LIN {X -0.304,Y -476.004,Z 243.555,A 0.000,B 0.000,C 90.000,E1 135.972} C_DIS
LIN {X 0.127,Y -476.516,Z 243.548,A 0.000,B 0.000,C 90.000,E1 134.676} C_DIS
LIN {X -0.220,Y -476.712,Z 243.543,A 0.000,B 0.000,C 90.000,E1 133.785} C_DIS
LIN {X -0.220,Y -476.693,Z 243.538,A 0.000,B 0.000,C 90.000,E1 132.852} C_DIS
LIN {X -0.114,Y -476.300,Z 243.531,A 0.000,B 0.000,C 90.000,E1 131.595} C_DIS
LIN {X 0.027,Y -475.504,Z 243.524,A 0.000,B 0.000,C 90.000,E1 130.334} C_DIS
LIN {X 0.251,Y -474.323,Z 243.515,A 0.000,B 0.000,C 90.000,E1 128.749} C_DIS
LIN {X -0.093,Y -473.444,Z 243.510,A 0.000,B 0.000,C 90.000,E1 127.855} C_DIS
LIN {X 0.085,Y -471.985,Z 243.503,A 0.000,B 0.000,C 90.000,E1 126.583} C_DIS
LIN {X 0.086,Y -470.799,Z 243.498,A 0.000,B 0.000,C 90.000,E1 125.644} C_DIS
LIN {X -0.119,Y -467.941,Z 243.488,A 0.000,B 0.000,C 90.000,E1 123.785} C_DIS
LIN {X 0.106,Y -465.899,Z 243.481,A 0.000,B 0.000,C 90.000,E1 122.498} C_DIS
LIN {X -0.098,Y -463.753,Z 243.474,A 0.000,B 0.000,C 90.000,E1 121.258} C_DIS
LIN {X -0.050,Y -461.019,Z 243.465,A 0.000,B 0.000,C 90.000,E1 119.667} C_DIS
LIN {X -0.164,Y -457.610,Z 243.454,A 0.000,B 0.000,C 90.000,E1 117.769} C_DIS
LIN {X -0.057,Y -454.742,Z 243.445,A 0.000,B 0.000,C 90.000,E1 116.155} C_DIS
LIN {X -0.026,Y -450.753,Z 243.433,A 0.000,B 0.000,C 90.000,E1 113.898} C_DIS
LIN {X -0.037,Y -449.140,Z 243.428,A 0.000,B 0.000,C 90.000,E1 112.950} C_DIS
LIN {X -0.075,Y -449.131,Z 243.428,A 0.000,B 0.000,C 90.000,E1 112.950} C_DIS
LIN {X 0.220,Y -456.665,Z 243.411,A 0.000,B 0.000,C 90.000,E1 109.993} C_DIS
LIN {X -0.034,Y -457.470,Z 243.410,A 0.000,B 0.000,C 90.000,E1 109.704} C_DIS
LIN {X 0.067,Y -466.135,Z 243.386,A 0.000,B 0.000,C 90.000,E1 105.552} C_DIS
LIN {X -0.209,Y -467.704,Z 243.383,A 0.000,B 0.000,C 90.000,E1 104.954} C_DIS
LIN {X 0.216,Y -475.915,Z 243.357,A 0.000,B 0.000,C 90.000,E1 100.197} C_DIS
LIN {X 0.055,Y -476.355,Z 243.355,A 0.000,B 0.000,C 90.000,E1 99.905} C_DIS
LIN {X 0.012,Y -481.875,Z 243.331,A 0.000,B 0.000,C 90.000,E1 95.568} C_DIS
LIN {X -0.141,Y -482.193,Z 243.329,A 0.000,B 0.000,C 90.000,E1 95.277} C_DIS
LIN {X -0.207,Y -485.365,Z 243.305,A 0.000,B 0.000,C 90.000,E1 90.974} C_DIS
LIN {X 0.102,Y -485.531,Z 243.304,A 0.000,B 0.000,C 90.000,E1 90.630} C_DIS
LIN {X -0.175,Y -486.345,Z 243.281,A 0.000,B 0.000,C 90.000,E1 86.674} C_DIS
LIN {X -0.041,Y -486.268,Z 243.278,A 0.000,B 0.000,C 90.000,E1 86.045} C_DIS
LIN {X 0.158,Y -484.694,Z 243.254,A 0.000,B 0.000,C 90.000,E1 81.724} C_DIS
LIN {X 0.026,Y -484.535,Z 243.252,A 0.000,B 0.000,C 90.000,E1 81.432} C_DIS
LIN {X -0.104,Y -480.473,Z 243.227,A 0.000,B 0.000,C 90.000,E1 76.825} C_DIS
LIN {X -0.207,Y -474.232,Z 243.201,A 0.000,B 0.000,C 90.000,E1 72.181} C_DIS
LIN {X 0.212,Y -473.736,Z 243.199,A 0.000,B 0.000,C 90.000,E1 71.819} C_DIS
LIN {X -0.275,Y -466.180,Z 243.175,A 0.000,B 0.000,C 90.000,E1 67.486} C_DIS
LIN {X 0.276,Y -465.753,Z 243.173,A 0.000,B 0.000,C 90.000,E1 67.102} C_DIS
LIN {X 0.046,Y -464.164,Z 243.169,A 0.000,B 0.000,C 90.000,E1 66.410} C_DIS
LIN {X 0.006,Y -464.156,Z 243.169,A 0.000,B 0.000,C 90.000,E1 66.410} C_DIS
LIN {X 0.084,Y -467.157,Z 243.162,A 0.000,B 0.000,C 90.000,E1 65.229} C_DIS
LIN {X 0.048,Y -470.372,Z 243.155,A 0.000,B 0.000,C 90.000,E1 63.973} C_DIS
LIN {X -0.028,Y -475.351,Z 243.145,A 0.000,B 0.000,C 90.000,E1 62.103} C_DIS
LIN {X 0.024,Y -481.156,Z 243.133,A 0.000,B 0.000,C 90.000,E1 59.921} C_DIS
LIN {X 0.004,Y -486.185,Z 243.123,A 0.000,B 0.000,C 90.000,E1 58.074} C_DIS
LIN {X -0.048,Y -490.388,Z 243.114,A 0.000,B 0.000,C 90.000,E1 56.548} C_DIS
LIN {X -0.011,Y -494.338,Z 243.106,A 0.000,B 0.000,C 90.000,E1 55.022} C_DIS
LIN {X -0.174,Y -497.233,Z 243.099,A 0.000,B 0.000,C 90.000,E1 53.829} C_DIS
LIN {X -0.174,Y -499.342,Z 243.094,A 0.000,B 0.000,C 90.000,E1 52.924} C_DIS
LIN {X 0.026,Y -501.806,Z 243.087,A 0.000,B 0.000,C 90.000,E1 51.698} C_DIS
LIN {X -0.131,Y -504.092,Z 243.081,A 0.000,B 0.000,C 90.000,E1 50.517} C_DIS
LIN {X -0.039,Y -506.583,Z 243.072,A 0.000,B 0.000,C 90.000,E1 49.013} C_DIS
LIN {X -0.178,Y -508.187,Z 243.066,A 0.000,B 0.000,C 90.000,E1 47.838} C_DIS
LIN {X -0.048,Y -508.957,Z 243.062,A 0.000,B 0.000,C 90.000,E1 47.229} C_DIS
LIN {X -0.149,Y -510.048,Z 243.056,A 0.000,B 0.000,C 90.000,E1 46.053} C_DIS
LIN {X 0.120,Y -510.862,Z 243.049,A 0.000,B 0.000,C 90.000,E1 44.838} C_DIS
LIN {X 0.048,Y -511.450,Z 243.043,A 0.000,B 0.000,C 90.000,E1 43.662} C_DIS
LIN {X 0.083,Y -511.654,Z 243.038,A 0.000,B 0.000,C 90.000,E1 42.771} C_DIS
LIN {X 0.018,Y -511.694,Z 243.031,A 0.000,B 0.000,C 90.000,E1 41.595} C_DIS
LIN {X -0.001,Y -511.374,Z 243.025,A 0.000,B 0.000,C 90.000,E1 40.415} C_DIS
LIN {X 0.309,Y -510.843,Z 243.018,A 0.000,B 0.000,C 90.000,E1 39.197} C_DIS
LIN {X 0.279,Y -509.901,Z 243.011,A 0.000,B 0.000,C 90.000,E1 38.016} C_DIS
LIN {X -0.079,Y -508.670,Z 243.005,A 0.000,B 0.000,C 90.000,E1 36.870} C_DIS
LIN {X -0.138,Y -506.605,Z 242.997,A 0.000,B 0.000,C 90.000,E1 35.391} C_DIS
LIN {X 0.072,Y -503.848,Z 242.987,A 0.000,B 0.000,C 90.000,E1 33.579} C_DIS
LIN {X 0.231,Y -500.339,Z 242.975,A 0.000,B 0.000,C 90.000,E1 31.465} C_DIS
LIN {X 0.059,Y -496.727,Z 242.962,A 0.000,B 0.000,C 90.000,E1 29.077} C_DIS
LIN {X -0.146,Y -492.657,Z 242.943,A 0.000,B 0.000,C 90.000,E1 25.771} C_DIS
LIN {X -0.140,Y -490.689,Z 242.931,A 0.000,B 0.000,C 90.000,E1 23.643} C_DIS
LIN {X 0.113,Y -488.478,Z 242.918,A 0.000,B 0.000,C 90.000,E1 21.173} C_DIS
LIN {X 0.135,Y -486.122,Z 242.902,A 0.000,B 0.000,C 90.000,E1 18.417} C_DIS
LIN {X 0.208,Y -484.424,Z 242.891,A 0.000,B 0.000,C 90.000,E1 16.260} C_DIS
LIN {X 0.101,Y -482.861,Z 242.879,A 0.000,B 0.000,C 90.000,E1 14.120} C_DIS
LIN {X -0.140,Y -481.824,Z 242.868,A 0.000,B 0.000,C 90.000,E1 12.299} C_DIS
LIN {X -0.164,Y -480.841,Z 242.856,A 0.000,B 0.000,C 90.000,E1 10.141} C_DIS
LIN {X 0.184,Y -480.149,Z 242.844,A 0.000,B 0.000,C 90.000,E1 7.936} C_DIS
LIN {X -0.241,Y -479.561,Z 242.831,A 0.000,B 0.000,C 90.000,E1 5.511} C_DIS
LIN {X 0.214,Y -479.518,Z 242.817,A 0.000,B 0.000,C 90.000,E1 2.980} C_DIS
LIN {X 0.105,Y -479.572,Z 242.812,A 0.000,B 0.000,C 90.000,E1 2.064} C_DIS
LIN {X 0.182,Y -480.137,Z 242.799,A 0.000,B 0.000,C 90.000,E1 359.771} C_DIS
LIN {X -0.082,Y -481.724,Z 242.783,A 0.000,B 0.000,C 90.000,E1 357.020} C_DIS
LIN {X 0.127,Y -483.318,Z 242.771,A 0.000,B 0.000,C 90.000,E1 354.837} C_DIS
LIN {X -0.041,Y -488.218,Z 242.748,A 0.000,B 0.000,C 90.000,E1 350.557} C_DIS
LIN {X 0.050,Y -492.322,Z 242.736,A 0.000,B 0.000,C 90.000,E1 348.409} C_DIS
LIN {X -0.131,Y -501.097,Z 242.717,A 0.000,B 0.000,C 90.000,E1 345.102} C_DIS
LIN {X 0.190,Y -506.043,Z 242.707,A 0.000,B 0.000,C 90.000,E1 343.268} C_DIS
LIN {X -0.058,Y -511.034,Z 242.697,A 0.000,B 0.000,C 90.000,E1 341.511} C_DIS
LIN {X -0.173,Y -521.016,Z 242.679,A 0.000,B 0.000,C 90.000,E1 338.284} C_DIS
LIN {X -0.192,Y -527.006,Z 242.670,A 0.000,B 0.000,C 90.000,E1 336.538} C_DIS
LIN {X -0.083,Y -533.082,Z 242.660,A 0.000,B 0.000,C 90.000,E1 334.793} C_DIS
LIN {X -0.107,Y -539.365,Z 242.650,A 0.000,B 0.000,C 90.000,E1 333.076} C_DIS
LIN {X -0.230,Y -545.756,Z 242.641,A 0.000,B 0.000,C 90.000,E1 331.385} C_DIS
LIN {X -0.216,Y -550.002,Z 242.635,A 0.000,B 0.000,C 90.000,E1 330.255} C_DIS
LIN {X 0.110,Y -555.145,Z 242.627,A 0.000,B 0.000,C 90.000,E1 328.820} C_DIS
LIN {X -0.088,Y -564.318,Z 242.613,A 0.000,B 0.000,C 90.000,E1 326.342} C_DIS
LIN {X 0.078,Y -571.677,Z 242.602,A 0.000,B 0.000,C 90.000,E1 324.402} C_DIS
LIN {X -0.167,Y -575.756,Z 242.596,A 0.000,B 0.000,C 90.000,E1 323.336} C_DIS
LIN {X -0.200,Y -580.262,Z 242.589,A 0.000,B 0.000,C 90.000,E1 321.984} C_DIS
LIN {X -0.276,Y -591.820,Z 242.571,A 0.000,B 0.000,C 90.000,E1 318.771} C_DIS
LIN {X 0.056,Y -596.053,Z 242.565,A 0.000,B 0.000,C 90.000,E1 317.676} C_DIS
LIN {X 0.042,Y -600.105,Z 242.559,A 0.000,B 0.000,C 90.000,E1 316.620} C_DIS
LIN {X 0.055,Y -603.953,Z 242.553,A 0.000,B 0.000,C 90.000,E1 315.567} C_DIS
LIN {X -0.066,Y -608.129,Z 242.546,A 0.000,B 0.000,C 90.000,E1 314.271} C_DIS
LIN {X 0.237,Y -610.253,Z 242.542,A 0.000,B 0.000,C 90.000,E1 313.461} C_DIS
LIN {X -0.035,Y -612.686,Z 242.536,A 0.000,B 0.000,C 90.000,E1 312.447} C_DIS
LIN {X 0.182,Y -614.592,Z 242.530,A 0.000,B 0.000,C 90.000,E1 311.391} C_DIS
LIN {X -0.036,Y -616.293,Z 242.524,A 0.000,B 0.000,C 90.000,E1 310.378} C_DIS
LIN {X 0.398,Y -617.459,Z 242.520,A 0.000,B 0.000,C 90.000,E1 309.564} C_DIS
LIN {X 0.291,Y -618.870,Z 242.514,A 0.000,B 0.000,C 90.000,E1 308.543} C_DIS
LIN {X 0.205,Y -620.140,Z 242.509,A 0.000,B 0.000,C 90.000,E1 307.523} C_DIS
LIN {X -0.193,Y -620.790,Z 242.504,A 0.000,B 0.000,C 90.000,E1 306.790} C_DIS
LIN {X -0.305,Y -621.404,Z 242.497,A 0.000,B 0.000,C 90.000,E1 305.518} C_DIS
LIN {X -0.197,Y -621.670,Z 242.493,A 0.000,B 0.000,C 90.000,E1 304.739} C_DIS
LIN {X 0.426,Y -621.842,Z 242.489,A 0.000,B 0.000,C 90.000,E1 303.913} C_DIS
LIN {X -0.348,Y -621.735,Z 242.483,A 0.000,B 0.000,C 90.000,E1 302.959} C_DIS
LIN {X 0.275,Y -621.168,Z 242.479,A 0.000,B 0.000,C 90.000,E1 302.133} C_DIS
LIN {X 0.018,Y -620.148,Z 242.473,A 0.000,B 0.000,C 90.000,E1 301.131} C_DIS
LIN {X 0.297,Y -619.048,Z 242.469,A 0.000,B 0.000,C 90.000,E1 300.335} C_DIS
LIN {X 0.010,Y -617.161,Z 242.463,A 0.000,B 0.000,C 90.000,E1 299.333} C_DIS
LIN {X -0.043,Y -615.539,Z 242.459,A 0.000,B 0.000,C 90.000,E1 298.565} C_DIS
LIN {X 0.129,Y -612.600,Z 242.452,A 0.000,B 0.000,C 90.000,E1 297.257} C_DIS
LIN {X 0.002,Y -609.954,Z 242.446,A 0.000,B 0.000,C 90.000,E1 296.232} C_DIS
LIN {X -0.210,Y -606.449,Z 242.439,A 0.000,B 0.000,C 90.000,E1 294.951} C_DIS
LIN {X -0.249,Y -602.264,Z 242.430,A 0.000,B 0.000,C 90.000,E1 293.387} C_DIS
LIN {X -0.218,Y -597.176,Z 242.418,A 0.000,B 0.000,C 90.000,E1 291.280} C_DIS
LIN {X 0.127,Y -592.982,Z 242.408,A 0.000,B 0.000,C 90.000,E1 289.396} C_DIS
LIN {X 0.188,Y -588.928,Z 242.398,A 0.000,B 0.000,C 90.000,E1 287.528} C_DIS
LIN {X 0.059,Y -584.239,Z 242.384,A 0.000,B 0.000,C 90.000,E1 285.134} C_DIS
LIN {X -0.183,Y -580.544,Z 242.372,A 0.000,B 0.000,C 90.000,E1 283.008} C_DIS
LIN {X -0.011,Y -576.449,Z 242.356,A 0.000,B 0.000,C 90.000,E1 280.018} C_DIS
LIN {X 0.186,Y -573.364,Z 242.339,A 0.000,B 0.000,C 90.000,E1 277.011} C_DIS
LIN {X 0.173,Y -571.959,Z 242.329,A 0.000,B 0.000,C 90.000,E1 275.106} C_DIS
LIN {X 0.208,Y -570.930,Z 242.297,A 0.000,B 0.000,C 90.000,E1 269.370} C_DIS
LIN {X -0.192,Y -574.912,Z 242.265,A 0.000,B 0.000,C 90.000,E1 263.685} C_DIS
LIN {X 0.272,Y -577.835,Z 242.251,A 0.000,B 0.000,C 90.000,E1 261.197} C_DIS
LIN {X 0.008,Y -581.772,Z 242.236,A 0.000,B 0.000,C 90.000,E1 258.522} C_DIS
LIN {X -0.055,Y -584.686,Z 242.226,A 0.000,B 0.000,C 90.000,E1 256.645} C_DIS
LIN {X 0.098,Y -585.933,Z 242.221,A 0.000,B 0.000,C 90.000,E1 255.825} C_DIS
LIN {X -0.236,Y -587.935,Z 242.214,A 0.000,B 0.000,C 90.000,E1 254.519} C_DIS
LIN {X -0.053,Y -589.315,Z 242.208,A 0.000,B 0.000,C 90.000,E1 253.433} C_DIS
LIN {X -0.121,Y -589.865,Z 242.205,A 0.000,B 0.000,C 90.000,E1 252.906} C_DIS
LIN {X -0.332,Y -590.543,Z 242.201,A 0.000,B 0.000,C 90.000,E1 252.127} C_DIS
LIN {X -0.109,Y -590.938,Z 242.195,A 0.000,B 0.000,C 90.000,E1 251.040} C_DIS
LIN {X 0.319,Y -591.095,Z 242.189,A 0.000,B 0.000,C 90.000,E1 249.934} C_DIS
LIN {X -0.007,Y -591.001,Z 242.183,A 0.000,B 0.000,C 90.000,E1 248.901} C_DIS
LIN {X -0.012,Y -590.558,Z 242.178,A 0.000,B 0.000,C 90.000,E1 248.103} C_DIS
LIN {X -0.026,Y -589.930,Z 242.174,A 0.000,B 0.000,C 90.000,E1 247.305} C_DIS
LIN {X 0.072,Y -588.643,Z 242.168,A 0.000,B 0.000,C 90.000,E1 246.230} C_DIS
LIN {X 0.273,Y -587.450,Z 242.164,A 0.000,B 0.000,C 90.000,E1 245.409} C_DIS
LIN {X 0.092,Y -585.402,Z 242.158,A 0.000,B 0.000,C 90.000,E1 244.357} C_DIS
LIN {X 0.257,Y -582.356,Z 242.150,A 0.000,B 0.000,C 90.000,E1 242.999} C_DIS
LIN {X -0.135,Y -578.999,Z 242.143,A 0.000,B 0.000,C 90.000,E1 241.691} C_DIS
LIN {X 0.076,Y -576.071,Z 242.137,A 0.000,B 0.000,C 90.000,E1 240.589} C_DIS
LIN {X -0.101,Y -573.711,Z 242.132,A 0.000,B 0.000,C 90.000,E1 239.793} C_DIS
LIN {X 0.255,Y -568.612,Z 242.123,A 0.000,B 0.000,C 90.000,E1 238.122} C_DIS
LIN {X -0.094,Y -564.190,Z 242.115,A 0.000,B 0.000,C 90.000,E1 236.786} C_DIS
LIN {X 0.047,Y -557.249,Z 242.103,A 0.000,B 0.000,C 90.000,E1 234.562} C_DIS
LIN {X -0.003,Y -552.836,Z 242.095,A 0.000,B 0.000,C 90.000,E1 233.176} C_DIS
LIN {X 0.027,Y -547.568,Z 242.086,A 0.000,B 0.000,C 90.000,E1 231.492} C_DIS
LIN {X -0.235,Y -542.222,Z 242.077,A 0.000,B 0.000,C 90.000,E1 229.828} C_DIS
LIN {X 0.163,Y -536.815,Z 242.067,A 0.000,B 0.000,C 90.000,E1 228.081} C_DIS
LIN {X 0.036,Y -531.322,Z 242.058,A 0.000,B 0.000,C 90.000,E1 226.377} C_DIS
LIN {X 0.198,Y -526.688,Z 242.050,A 0.000,B 0.000,C 90.000,E1 224.919} C_DIS
LIN {X -0.164,Y -521.139,Z 242.040,A 0.000,B 0.000,C 90.000,E1 223.218} C_DIS
LIN {X 0.033,Y -514.869,Z 242.029,A 0.000,B 0.000,C 90.000,E1 221.148} C_DIS
LIN {X 0.129,Y -508.712,Z 242.017,A 0.000,B 0.000,C 90.000,E1 219.072} C_DIS
LIN {X 0.060,Y -502.784,Z 242.006,A 0.000,B 0.000,C 90.000,E1 216.996} C_DIS
LIN {X 0.160,Y -497.674,Z 241.996,A 0.000,B 0.000,C 90.000,E1 215.185} C_DIS
LIN {X -0.109,Y -493.403,Z 241.987,A 0.000,B 0.000,C 90.000,E1 213.706} C_DIS
LIN {X -0.072,Y -488.405,Z 241.977,A 0.000,B 0.000,C 90.000,E1 211.878} C_DIS
LIN {X -0.168,Y -482.790,Z 241.965,A 0.000,B 0.000,C 90.000,E1 209.745} C_DIS
LIN {X -0.152,Y -474.126,Z 241.945,A 0.000,B 0.000,C 90.000,E1 206.027} C_DIS
LIN {X -0.023,Y -469.618,Z 241.932,A 0.000,B 0.000,C 90.000,E1 203.823} C_DIS
LIN {X -0.251,Y -462.865,Z 241.911,A 0.000,B 0.000,C 90.000,E1 200.066} C_DIS
LIN {X -0.040,Y -458.061,Z 241.894,A 0.000,B 0.000,C 90.000,E1 196.858} C_DIS
LIN {X 0.143,Y -454.256,Z 241.878,A 0.000,B 0.000,C 90.000,E1 193.953} C_DIS
LIN {X 0.059,Y -452.251,Z 241.869,A 0.000,B 0.000,C 90.000,E1 192.355} C_DIS
LIN {X -0.106,Y -449.238,Z 241.854,A 0.000,B 0.000,C 90.000,E1 189.792} C_DIS
LIN {X 0.010,Y -446.505,Z 241.840,A 0.000,B 0.000,C 90.000,E1 187.182} C_DIS
LIN {X 0.200,Y -444.448,Z 241.827,A 0.000,B 0.000,C 90.000,E1 184.878} C_DIS
LIN {X -0.109,Y -443.337,Z 241.820,A 0.000,B 0.000,C 90.000,E1 183.612} C_DIS
LIN {X -0.022,Y -442.321,Z 241.813,A 0.000,B 0.000,C 90.000,E1 182.293} C_DIS
LIN {X 0.169,Y -441.174,Z 241.804,A 0.000,B 0.000,C 90.000,E1 180.630} C_DIS
LIN {X -0.190,Y -439.660,Z 241.789,A 0.000,B 0.000,C 90.000,E1 178.051} C_DIS
LIN {X 0.101,Y -438.687,Z 241.771,A 0.000,B 0.000,C 90.000,E1 174.723} C_DIS
LIN {X -0.213,Y -438.624,Z 241.751,A 0.000,B 0.000,C 90.000,E1 171.141} C_DIS
LIN {X 0.102,Y -439.157,Z 241.736,A 0.000,B 0.000,C 90.000,E1 168.465} C_DIS
LIN {X -0.031,Y -440.655,Z 241.716,A 0.000,B 0.000,C 90.000,E1 164.866} C_DIS
LIN {X 0.008,Y -441.997,Z 241.701,A 0.000,B 0.000,C 90.000,E1 162.236} C_DIS
LIN {X 0.086,Y -443.455,Z 241.689,A 0.000,B 0.000,C 90.000,E1 159.934} C_DIS
LIN {X 0.076,Y -446.041,Z 241.672,A 0.000,B 0.000,C 90.000,E1 156.997} C_DIS
LIN {X 0.106,Y -448.492,Z 241.660,A 0.000,B 0.000,C 90.000,E1 154.717} C_DIS
LIN {X -0.112,Y -451.766,Z 241.645,A 0.000,B 0.000,C 90.000,E1 152.153} C_DIS
LIN {X 0.095,Y -455.084,Z 241.633,A 0.000,B 0.000,C 90.000,E1 149.871} C_DIS
LIN {X -0.173,Y -458.625,Z 241.620,A 0.000,B 0.000,C 90.000,E1 147.661} C_DIS
LIN {X 0.151,Y -462.336,Z 241.608,A 0.000,B 0.000,C 90.000,E1 145.388} C_DIS
LIN {X -0.075,Y -464.957,Z 241.599,A 0.000,B 0.000,C 90.000,E1 143.829} C_DIS
LIN {X -0.255,Y -467.359,Z 241.590,A 0.000,B 0.000,C 90.000,E1 142.271} C_DIS
LIN {X -0.048,Y -470.004,Z 241.580,A 0.000,B 0.000,C 90.000,E1 140.356} C_DIS
LIN {X 0.082,Y -471.957,Z 241.571,A 0.000,B 0.000,C 90.000,E1 138.771} C_DIS
LIN {X -0.199,Y -473.178,Z 241.564,A 0.000,B 0.000,C 90.000,E1 137.553} C_DIS
LIN {X -0.144,Y -474.125,Z 241.557,A 0.000,B 0.000,C 90.000,E1 136.296} C_DIS
LIN {X 0.054,Y -474.411,Z 241.554,A 0.000,B 0.000,C 90.000,E1 135.648} C_DIS
LIN {X 0.256,Y -474.787,Z 241.550,A 0.000,B 0.000,C 90.000,E1 135.000} C_DIS
LIN {X -0.007,Y -475.074,Z 241.543,A 0.000,B 0.000,C 90.000,E1 133.785} C_DIS
LIN {X -0.026,Y -475.093,Z 241.538,A 0.000,B 0.000,C 90.000,E1 132.852} C_DIS
LIN {X 0.055,Y -474.641,Z 241.531,A 0.000,B 0.000,C 90.000,E1 131.595} C_DIS
LIN {X 0.260,Y -473.640,Z 241.523,A 0.000,B 0.000,C 90.000,E1 130.011} C_DIS
LIN {X -0.304,Y -472.672,Z 241.516,A 0.000,B 0.000,C 90.000,E1 128.830} C_DIS
LIN {X 0.000,Y -471.795,Z 241.510,A 0.000,B 0.000,C 90.000,E1 127.855} C_DIS
LIN {X 0.152,Y -470.389,Z 241.503,A 0.000,B 0.000,C 90.000,E1 126.583} C_DIS
LIN {X -0.095,Y -468.779,Z 241.496,A 0.000,B 0.000,C 90.000,E1 125.358} C_DIS
LIN {X 0.043,Y -465.891,Z 241.486,A 0.000,B 0.000,C 90.000,E1 123.452} C_DIS
LIN {X -0.154,Y -463.815,Z 241.479,A 0.000,B 0.000,C 90.000,E1 122.212} C_DIS
LIN {X 0.002,Y -461.640,Z 241.472,A 0.000,B 0.000,C 90.000,E1 120.924} C_DIS
LIN {X 0.008,Y -458.916,Z 241.463,A 0.000,B 0.000,C 90.000,E1 119.333} C_DIS
LIN {X 0.140,Y -456.050,Z 241.454,A 0.000,B 0.000,C 90.000,E1 117.719} C_DIS
LIN {X 0.110,Y -452.565,Z 241.443,A 0.000,B 0.000,C 90.000,E1 115.796} C_DIS
LIN {X -0.137,Y -448.627,Z 241.431,A 0.000,B 0.000,C 90.000,E1 113.567} C_DIS
LIN {X -0.056,Y -448.249,Z 241.430,A 0.000,B 0.000,C 90.000,E1 113.334} C_DIS
LIN {X -0.096,Y -448.253,Z 241.430,A 0.000,B 0.000,C 90.000,E1 113.334} C_DIS
LIN {X 0.025,Y -456.735,Z 241.411,A 0.000,B 0.000,C 90.000,E1 109.993} C_DIS
LIN {X -0.074,Y -457.513,Z 241.409,A 0.000,B 0.000,C 90.000,E1 109.685} C_DIS
LIN {X -0.129,Y -466.192,Z 241.386,A 0.000,B 0.000,C 90.000,E1 105.552} C_DIS
LIN {X 0.048,Y -467.758,Z 241.383,A 0.000,B 0.000,C 90.000,E1 104.898} C_DIS
LIN {X 0.020,Y -475.965,Z 241.357,A 0.000,B 0.000,C 90.000,E1 100.197} C_DIS
LIN {X 0.169,Y -476.677,Z 241.353,A 0.000,B 0.000,C 90.000,E1 99.557} C_DIS
LIN {X -0.186,Y -481.913,Z 241.331,A 0.000,B 0.000,C 90.000,E1 95.568} C_DIS
LIN {X 0.142,Y -482.202,Z 241.329,A 0.000,B 0.000,C 90.000,E1 95.220} C_DIS
LIN {X 0.080,Y -485.389,Z 241.305,A 0.000,B 0.000,C 90.000,E1 90.917} C_DIS
LIN {X -0.096,Y -485.529,Z 241.303,A 0.000,B 0.000,C 90.000,E1 90.630} C_DIS
LIN {X 0.113,Y -486.357,Z 241.281,A 0.000,B 0.000,C 90.000,E1 86.617} C_DIS
LIN {X -0.063,Y -486.368,Z 241.280,A 0.000,B 0.000,C 90.000,E1 86.331} C_DIS
LIN {X -0.074,Y -485.858,Z 241.275,A 0.000,B 0.000,C 90.000,E1 85.412} C_DIS
LIN {X -0.039,Y -484.692,Z 241.254,A 0.000,B 0.000,C 90.000,E1 81.724} C_DIS
LIN {X -0.171,Y -484.506,Z 241.252,A 0.000,B 0.000,C 90.000,E1 81.432} C_DIS
LIN {X 0.167,Y -480.439,Z 241.227,A 0.000,B 0.000,C 90.000,E1 76.769} C_DIS
LIN {X 0.049,Y -474.209,Z 241.201,A 0.000,B 0.000,C 90.000,E1 72.127} C_DIS
LIN {X -0.017,Y -473.050,Z 241.197,A 0.000,B 0.000,C 90.000,E1 71.511} C_DIS
LIN {X 0.081,Y -465.722,Z 241.173,A 0.000,B 0.000,C 90.000,E1 67.102} C_DIS
LIN {X -0.052,Y -463.440,Z 241.167,A 0.000,B 0.000,C 90.000,E1 66.102} C_DIS
LIN {X -0.092,Y -463.437,Z 241.167,A 0.000,B 0.000,C 90.000,E1 66.102} C_DIS
LIN {X -0.056,Y -467.282,Z 241.159,A 0.000,B 0.000,C 90.000,E1 64.588} C_DIS
LIN {X 0.174,Y -473.040,Z 241.147,A 0.000,B 0.000,C 90.000,E1 62.359} C_DIS
LIN {X -0.025,Y -477.955,Z 241.136,A 0.000,B 0.000,C 90.000,E1 60.511} C_DIS
LIN {X -0.120,Y -481.302,Z 241.129,A 0.000,B 0.000,C 90.000,E1 59.282} C_DIS
LIN {X 0.105,Y -486.372,Z 241.119,A 0.000,B 0.000,C 90.000,E1 57.406} C_DIS
LIN {X -0.187,Y -489.686,Z 241.112,A 0.000,B 0.000,C 90.000,E1 56.215} C_DIS
LIN {X -0.016,Y -492.807,Z 241.105,A 0.000,B 0.000,C 90.000,E1 54.975} C_DIS
LIN {X -0.055,Y -496.411,Z 241.097,A 0.000,B 0.000,C 90.000,E1 53.463} C_DIS
LIN {X -0.063,Y -498.422,Z 241.092,A 0.000,B 0.000,C 90.000,E1 52.557} C_DIS
LIN {X 0.124,Y -500.820,Z 241.085,A 0.000,B 0.000,C 90.000,E1 51.331} C_DIS
LIN {X -0.049,Y -502.956,Z 241.079,A 0.000,B 0.000,C 90.000,E1 50.150} C_DIS
LIN {X 0.019,Y -505.388,Z 241.070,A 0.000,B 0.000,C 90.000,E1 48.647} C_DIS
LIN {X -0.138,Y -506.930,Z 241.064,A 0.000,B 0.000,C 90.000,E1 47.472} C_DIS
LIN {X -0.270,Y -508.199,Z 241.057,A 0.000,B 0.000,C 90.000,E1 46.296} C_DIS
LIN {X -0.031,Y -509.037,Z 241.050,A 0.000,B 0.000,C 90.000,E1 45.081} C_DIS
LIN {X 0.223,Y -509.627,Z 241.044,A 0.000,B 0.000,C 90.000,E1 43.866} C_DIS
LIN {X -0.114,Y -509.883,Z 241.039,A 0.000,B 0.000,C 90.000,E1 43.014} C_DIS
LIN {X -0.203,Y -509.929,Z 241.032,A 0.000,B 0.000,C 90.000,E1 41.838} C_DIS
LIN {X 0.182,Y -509.786,Z 241.027,A 0.000,B 0.000,C 90.000,E1 40.906} C_DIS
LIN {X 0.230,Y -509.425,Z 241.022,A 0.000,B 0.000,C 90.000,E1 40.011} C_DIS
LIN {X 0.274,Y -508.952,Z 241.018,A 0.000,B 0.000,C 90.000,E1 39.116} C_DIS
LIN {X -0.098,Y -508.008,Z 241.011,A 0.000,B 0.000,C 90.000,E1 37.971} C_DIS
LIN {X 0.136,Y -506.244,Z 241.003,A 0.000,B 0.000,C 90.000,E1 36.457} C_DIS
LIN {X -0.073,Y -503.631,Z 240.993,A 0.000,B 0.000,C 90.000,E1 34.692} C_DIS
LIN {X -0.182,Y -503.022,Z 240.991,A 0.000,B 0.000,C 90.000,E1 34.405} C_DIS
LIN {X 0.187,Y -501.173,Z 240.984,A 0.000,B 0.000,C 90.000,E1 33.166} C_DIS
LIN {X -0.038,Y -499.532,Z 240.979,A 0.000,B 0.000,C 90.000,E1 32.291} C_DIS
LIN {X -0.017,Y -498.078,Z 240.974,A 0.000,B 0.000,C 90.000,E1 31.386} C_DIS
LIN {X -0.249,Y -496.160,Z 240.968,A 0.000,B 0.000,C 90.000,E1 30.207} C_DIS
LIN {X -0.099,Y -494.888,Z 240.963,A 0.000,B 0.000,C 90.000,E1 29.283} C_DIS
LIN {X -0.109,Y -492.765,Z 240.954,A 0.000,B 0.000,C 90.000,E1 27.769} C_DIS
LIN {X -0.071,Y -489.839,Z 240.939,A 0.000,B 0.000,C 90.000,E1 25.027} C_DIS
LIN {X -0.130,Y -488.013,Z 240.927,A 0.000,B 0.000,C 90.000,E1 22.898} C_DIS
LIN {X 0.040,Y -485.827,Z 240.914,A 0.000,B 0.000,C 90.000,E1 20.429} C_DIS
LIN {X -0.196,Y -483.497,Z 240.898,A 0.000,B 0.000,C 90.000,E1 17.692} C_DIS
LIN {X -0.040,Y -482.334,Z 240.890,A 0.000,B 0.000,C 90.000,E1 16.134} C_DIS
LIN {X -0.173,Y -480.268,Z 240.873,A 0.000,B 0.000,C 90.000,E1 13.063} C_DIS
LIN {X 0.145,Y -479.410,Z 240.864,A 0.000,B 0.000,C 90.000,E1 11.478} C_DIS
LIN {X 0.204,Y -478.656,Z 240.854,A 0.000,B 0.000,C 90.000,E1 9.613} C_DIS
LIN {X 0.164,Y -478.115,Z 240.843,A 0.000,B 0.000,C 90.000,E1 7.757} C_DIS
LIN {X 0.141,Y -477.572,Z 240.829,A 0.000,B 0.000,C 90.000,E1 5.277} C_DIS
LIN {X 0.224,Y -477.544,Z 240.817,A 0.000,B 0.000,C 90.000,E1 3.094} C_DIS
LIN {X -0.109,Y -477.629,Z 240.810,A 0.000,B 0.000,C 90.000,E1 1.892} C_DIS
LIN {X -0.036,Y -479.160,Z 240.789,A 0.000,B 0.000,C 90.000,E1 357.936} C_DIS
LIN {X 0.081,Y -480.630,Z 240.777,A 0.000,B 0.000,C 90.000,E1 355.755} C_DIS
LIN {X 0.089,Y -486.730,Z 240.746,A 0.000,B 0.000,C 90.000,E1 350.208} C_DIS
LIN {X -0.230,Y -490.366,Z 240.736,A 0.000,B 0.000,C 90.000,E1 348.409} C_DIS
LIN {X 0.072,Y -498.285,Z 240.719,A 0.000,B 0.000,C 90.000,E1 345.338} C_DIS
LIN {X -0.072,Y -502.416,Z 240.710,A 0.000,B 0.000,C 90.000,E1 343.850} C_DIS
LIN {X -0.147,Y -506.534,Z 240.702,A 0.000,B 0.000,C 90.000,E1 342.362} C_DIS
LIN {X 0.150,Y -513.432,Z 240.689,A 0.000,B 0.000,C 90.000,E1 339.953} C_DIS
LIN {X -0.143,Y -523.090,Z 240.672,A 0.000,B 0.000,C 90.000,E1 337.050} C_DIS
LIN {X 0.275,Y -530.175,Z 240.661,A 0.000,B 0.000,C 90.000,E1 334.973} C_DIS
LIN {X 0.002,Y -535.343,Z 240.653,A 0.000,B 0.000,C 90.000,E1 333.563} C_DIS
LIN {X 0.030,Y -541.740,Z 240.644,A 0.000,B 0.000,C 90.000,E1 331.847} C_DIS
LIN {X -0.268,Y -547.148,Z 240.636,A 0.000,B 0.000,C 90.000,E1 330.461} C_DIS
LIN {X -0.231,Y -551.301,Z 240.630,A 0.000,B 0.000,C 90.000,E1 329.331} C_DIS
LIN {X -0.302,Y -557.370,Z 240.620,A 0.000,B 0.000,C 90.000,E1 327.661} C_DIS
LIN {X 0.147,Y -564.644,Z 240.609,A 0.000,B 0.000,C 90.000,E1 325.674} C_DIS
LIN {X -0.075,Y -569.948,Z 240.602,A 0.000,B 0.000,C 90.000,E1 324.322} C_DIS
LIN {X 0.118,Y -573.994,Z 240.596,A 0.000,B 0.000,C 90.000,E1 323.210} C_DIS
LIN {X 0.251,Y -577.673,Z 240.590,A 0.000,B 0.000,C 90.000,E1 322.110} C_DIS
LIN {X -0.038,Y -588.258,Z 240.573,A 0.000,B 0.000,C 90.000,E1 319.175} C_DIS
LIN {X 0.200,Y -594.599,Z 240.564,A 0.000,B 0.000,C 90.000,E1 317.553} C_DIS
LIN {X -0.275,Y -598.706,Z 240.558,A 0.000,B 0.000,C 90.000,E1 316.539} C_DIS
LIN {X -0.283,Y -602.524,Z 240.553,A 0.000,B 0.000,C 90.000,E1 315.486} C_DIS
LIN {X -0.235,Y -605.841,Z 240.547,A 0.000,B 0.000,C 90.000,E1 314.433} C_DIS
LIN {X 0.234,Y -607.417,Z 240.544,A 0.000,B 0.000,C 90.000,E1 313.866} C_DIS
LIN {X -0.073,Y -610.076,Z 240.538,A 0.000,B 0.000,C 90.000,E1 312.852} C_DIS
LIN {X -0.346,Y -612.139,Z 240.532,A 0.000,B 0.000,C 90.000,E1 311.838} C_DIS
LIN {X -0.135,Y -613.846,Z 240.527,A 0.000,B 0.000,C 90.000,E1 310.782} C_DIS
LIN {X 0.103,Y -615.379,Z 240.521,A 0.000,B 0.000,C 90.000,E1 309.725} C_DIS
LIN {X -0.030,Y -616.752,Z 240.515,A 0.000,B 0.000,C 90.000,E1 308.705} C_DIS
LIN {X 0.237,Y -618.048,Z 240.509,A 0.000,B 0.000,C 90.000,E1 307.649} C_DIS
LIN {X 0.311,Y -618.713,Z 240.505,A 0.000,B 0.000,C 90.000,E1 306.870} C_DIS
LIN {X -0.151,Y -619.223,Z 240.499,A 0.000,B 0.000,C 90.000,E1 305.884} C_DIS
LIN {X -0.287,Y -619.733,Z 240.492,A 0.000,B 0.000,C 90.000,E1 304.612} C_DIS
LIN {X -0.198,Y -619.874,Z 240.488,A 0.000,B 0.000,C 90.000,E1 303.833} C_DIS
LIN {X 0.063,Y -619.738,Z 240.484,A 0.000,B 0.000,C 90.000,E1 303.038} C_DIS
LIN {X -0.166,Y -619.560,Z 240.481,A 0.000,B 0.000,C 90.000,E1 302.546} C_DIS
LIN {X -0.139,Y -618.378,Z 240.474,A 0.000,B 0.000,C 90.000,E1 301.258} C_DIS
LIN {X 0.080,Y -616.402,Z 240.466,A 0.000,B 0.000,C 90.000,E1 299.951} C_DIS
LIN {X -0.215,Y -614.887,Z 240.462,A 0.000,B 0.000,C 90.000,E1 299.205} C_DIS
LIN {X -0.056,Y -612.133,Z 240.455,A 0.000,B 0.000,C 90.000,E1 297.897} C_DIS
LIN {X -0.154,Y -610.316,Z 240.451,A 0.000,B 0.000,C 90.000,E1 297.129} C_DIS
LIN {X 0.144,Y -606.243,Z 240.442,A 0.000,B 0.000,C 90.000,E1 295.540} C_DIS
LIN {X -0.131,Y -602.752,Z 240.435,A 0.000,B 0.000,C 90.000,E1 294.259} C_DIS
LIN {X -0.026,Y -595.559,Z 240.419,A 0.000,B 0.000,C 90.000,E1 291.354} C_DIS
LIN {X 0.045,Y -591.964,Z 240.410,A 0.000,B 0.000,C 90.000,E1 289.758} C_DIS
LIN {X 0.260,Y -587.932,Z 240.399,A 0.000,B 0.000,C 90.000,E1 287.873} C_DIS
LIN {X 0.081,Y -583.150,Z 240.386,A 0.000,B 0.000,C 90.000,E1 285.481} C_DIS
LIN {X 0.021,Y -578.935,Z 240.373,A 0.000,B 0.000,C 90.000,E1 283.063} C_DIS
LIN {X 0.228,Y -574.455,Z 240.355,A 0.000,B 0.000,C 90.000,E1 279.792} C_DIS
LIN {X 0.249,Y -571.636,Z 240.339,A 0.000,B 0.000,C 90.000,E1 277.068} C_DIS
LIN {X 0.157,Y -569.586,Z 240.323,A 0.000,B 0.000,C 90.000,E1 274.073} C_DIS
LIN {X -0.032,Y -569.074,Z 240.298,A 0.000,B 0.000,C 90.000,E1 269.714} C_DIS
LIN {X 0.133,Y -573.052,Z 240.265,A 0.000,B 0.000,C 90.000,E1 263.685} C_DIS
LIN {X 0.132,Y -575.300,Z 240.254,A 0.000,B 0.000,C 90.000,E1 261.781} C_DIS
LIN {X -0.095,Y -578.217,Z 240.242,A 0.000,B 0.000,C 90.000,E1 259.634} C_DIS
LIN {X -0.132,Y -580.308,Z 240.235,A 0.000,B 0.000,C 90.000,E1 258.285} C_DIS
LIN {X -0.228,Y -583.304,Z 240.224,A 0.000,B 0.000,C 90.000,E1 256.408} C_DIS
LIN {X -0.035,Y -585.341,Z 240.217,A 0.000,B 0.000,C 90.000,E1 255.046} C_DIS
LIN {X 0.191,Y -587.211,Z 240.210,A 0.000,B 0.000,C 90.000,E1 253.685} C_DIS
LIN {X 0.276,Y -587.874,Z 240.207,A 0.000,B 0.000,C 90.000,E1 253.142} C_DIS
LIN {X -0.276,Y -588.783,Z 240.201,A 0.000,B 0.000,C 90.000,E1 252.127} C_DIS
LIN {X 0.247,Y -589.132,Z 240.196,A 0.000,B 0.000,C 90.000,E1 251.275} C_DIS
LIN {X -0.104,Y -589.338,Z 240.190,A 0.000,B 0.000,C 90.000,E1 250.242} C_DIS
LIN {X 0.098,Y -589.281,Z 240.184,A 0.000,B 0.000,C 90.000,E1 249.156} C_DIS
LIN {X -0.142,Y -589.165,Z 240.181,A 0.000,B 0.000,C 90.000,E1 248.646} C_DIS
LIN {X 0.265,Y -588.403,Z 240.175,A 0.000,B 0.000,C 90.000,E1 247.539} C_DIS
LIN {X 0.229,Y -587.595,Z 240.171,A 0.000,B 0.000,C 90.000,E1 246.741} C_DIS
LIN {X -0.121,Y -586.552,Z 240.167,A 0.000,B 0.000,C 90.000,E1 245.973} C_DIS
LIN {X 0.060,Y -585.187,Z 240.162,A 0.000,B 0.000,C 90.000,E1 245.153} C_DIS
LIN {X 0.226,Y -583.623,Z 240.158,A 0.000,B 0.000,C 90.000,E1 244.332} C_DIS
LIN {X -0.150,Y -581.816,Z 240.153,A 0.000,B 0.000,C 90.000,E1 243.563} C_DIS
LIN {X -0.163,Y -579.212,Z 240.147,A 0.000,B 0.000,C 90.000,E1 242.487} C_DIS
LIN {X 0.048,Y -576.413,Z 240.141,A 0.000,B 0.000,C 90.000,E1 241.385} C_DIS
LIN {X -0.286,Y -573.354,Z 240.135,A 0.000,B 0.000,C 90.000,E1 240.333} C_DIS
LIN {X 0.001,Y -570.932,Z 240.131,A 0.000,B 0.000,C 90.000,E1 239.488} C_DIS
LIN {X -0.197,Y -565.853,Z 240.121,A 0.000,B 0.000,C 90.000,E1 237.867} C_DIS
LIN {X 0.020,Y -564.026,Z 240.118,A 0.000,B 0.000,C 90.000,E1 237.296} C_DIS
LIN {X -0.181,Y -563.262,Z 240.117,A 0.000,B 0.000,C 90.000,E1 237.041} C_DIS
LIN {X -0.287,Y -561.375,Z 240.114,A 0.000,B 0.000,C 90.000,E1 236.501} C_DIS
LIN {X -0.227,Y -557.963,Z 240.108,A 0.000,B 0.000,C 90.000,E1 235.388} C_DIS
LIN {X -0.142,Y -553.628,Z 240.100,A 0.000,B 0.000,C 90.000,E1 233.989} C_DIS
LIN {X 0.127,Y -549.989,Z 240.094,A 0.000,B 0.000,C 90.000,E1 232.844} C_DIS
LIN {X -0.088,Y -546.541,Z 240.087,A 0.000,B 0.000,C 90.000,E1 231.743} C_DIS
LIN {X 0.071,Y -542.920,Z 240.081,A 0.000,B 0.000,C 90.000,E1 230.598} C_DIS
LIN {X 0.100,Y -539.387,Z 240.075,A 0.000,B 0.000,C 90.000,E1 229.461} C_DIS
LIN {X 0.076,Y -534.850,Z 240.067,A 0.000,B 0.000,C 90.000,E1 228.038} C_DIS
LIN {X -0.071,Y -530.240,Z 240.059,A 0.000,B 0.000,C 90.000,E1 226.620} C_DIS
LIN {X 0.015,Y -524.601,Z 240.049,A 0.000,B 0.000,C 90.000,E1 224.879} C_DIS
LIN {X 0.128,Y -520.919,Z 240.043,A 0.000,B 0.000,C 90.000,E1 223.704} C_DIS
LIN {X -0.142,Y -513.690,Z 240.030,A 0.000,B 0.000,C 90.000,E1 221.391} C_DIS
LIN {X 0.157,Y -506.625,Z 240.017,A 0.000,B 0.000,C 90.000,E1 218.991} C_DIS
LIN {X -0.270,Y -500.706,Z 240.005,A 0.000,B 0.000,C 90.000,E1 216.950} C_DIS
LIN {X 0.082,Y -495.605,Z 239.995,A 0.000,B 0.000,C 90.000,E1 215.105} C_DIS
LIN {X -0.132,Y -489.669,Z 239.983,A 0.000,B 0.000,C 90.000,E1 213.007} C_DIS
LIN {X 0.229,Y -484.652,Z 239.973,A 0.000,B 0.000,C 90.000,E1 211.131} C_DIS
LIN {X 0.023,Y -479.055,Z 239.961,A 0.000,B 0.000,C 90.000,E1 208.999} C_DIS
LIN {X -0.062,Y -471.973,Z 239.944,A 0.000,B 0.000,C 90.000,E1 205.899} C_DIS
LIN {X -0.045,Y -466.911,Z 239.930,A 0.000,B 0.000,C 90.000,E1 203.387} C_DIS
LIN {X 0.114,Y -460.821,Z 239.911,A 0.000,B 0.000,C 90.000,E1 199.885} C_DIS
LIN {X 0.244,Y -456.102,Z 239.893,A 0.000,B 0.000,C 90.000,E1 196.677} C_DIS
LIN {X -0.088,Y -452.308,Z 239.877,A 0.000,B 0.000,C 90.000,E1 193.828} C_DIS
LIN {X 0.130,Y -450.288,Z 239.868,A 0.000,B 0.000,C 90.000,E1 192.187} C_DIS
LIN {X -0.009,Y -447.293,Z 239.853,A 0.000,B 0.000,C 90.000,E1 189.613} C_DIS
LIN {X 0.035,Y -444.568,Z 239.839,A 0.000,B 0.000,C 90.000,E1 187.004} C_DIS
LIN {X 0.160,Y -442.532,Z 239.826,A 0.000,B 0.000,C 90.000,E1 184.702} C_DIS
LIN {X 0.050,Y -440.960,Z 239.815,A 0.000,B 0.000,C 90.000,E1 182.751} C_DIS
LIN {X 0.001,Y -439.256,Z 239.803,A 0.000,B 0.000,C 90.000,E1 180.458} C_DIS
LIN {X -0.206,Y -437.500,Z 239.784,A 0.000,B 0.000,C 90.000,E1 177.192} C_DIS
LIN {X 0.062,Y -436.786,Z 239.766,A 0.000,B 0.000,C 90.000,E1 173.856} C_DIS
LIN {X 0.036,Y -436.965,Z 239.748,A 0.000,B 0.000,C 90.000,E1 170.557} C_DIS
LIN {X -0.129,Y -437.553,Z 239.733,A 0.000,B 0.000,C 90.000,E1 167.937} C_DIS
LIN {X 0.134,Y -438.835,Z 239.716,A 0.000,B 0.000,C 90.000,E1 164.936} C_DIS
LIN {X -0.024,Y -440.012,Z 239.704,A 0.000,B 0.000,C 90.000,E1 162.653} C_DIS
LIN {X -0.030,Y -441.908,Z 239.687,A 0.000,B 0.000,C 90.000,E1 159.699} C_DIS
LIN {X 0.208,Y -444.230,Z 239.673,A 0.000,B 0.000,C 90.000,E1 157.050} C_DIS
LIN {X 0.004,Y -446.687,Z 239.660,A 0.000,B 0.000,C 90.000,E1 154.793} C_DIS
LIN {X -0.281,Y -449.913,Z 239.646,A 0.000,B 0.000,C 90.000,E1 152.231} C_DIS
LIN {X 0.093,Y -453.248,Z 239.633,A 0.000,B 0.000,C 90.000,E1 149.921} C_DIS
LIN {X -0.106,Y -457.311,Z 239.619,A 0.000,B 0.000,C 90.000,E1 147.375} C_DIS
LIN {X 0.186,Y -461.031,Z 239.606,A 0.000,B 0.000,C 90.000,E1 145.102} C_DIS
LIN {X -0.062,Y -463.671,Z 239.597,A 0.000,B 0.000,C 90.000,E1 143.543} C_DIS
LIN {X 0.020,Y -466.095,Z 239.589,A 0.000,B 0.000,C 90.000,E1 141.949} C_DIS
LIN {X 0.143,Y -468.307,Z 239.580,A 0.000,B 0.000,C 90.000,E1 140.356} C_DIS
LIN {X 0.240,Y -470.195,Z 239.571,A 0.000,B 0.000,C 90.000,E1 138.771} C_DIS
LIN {X -0.066,Y -471.507,Z 239.564,A 0.000,B 0.000,C 90.000,E1 137.553} C_DIS
LIN {X -0.038,Y -472.398,Z 239.557,A 0.000,B 0.000,C 90.000,E1 136.296} C_DIS
LIN {X -0.240,Y -473.142,Z 239.549,A 0.000,B 0.000,C 90.000,E1 134.757} C_DIS
LIN {X 0.046,Y -473.344,Z 239.543,A 0.000,B 0.000,C 90.000,E1 133.785} C_DIS
LIN {X 0.102,Y -473.269,Z 239.536,A 0.000,B 0.000,C 90.000,E1 132.528} C_DIS
LIN {X 0.062,Y -472.878,Z 239.531,A 0.000,B 0.000,C 90.000,E1 131.595} C_DIS
LIN {X 0.234,Y -471.967,Z 239.522,A 0.000,B 0.000,C 90.000,E1 130.011} C_DIS
LIN {X 0.086,Y -470.722,Z 239.514,A 0.000,B 0.000,C 90.000,E1 128.463} C_DIS
LIN {X 0.283,Y -469.143,Z 239.505,A 0.000,B 0.000,C 90.000,E1 126.870} C_DIS
LIN {X 0.166,Y -467.160,Z 239.496,A 0.000,B 0.000,C 90.000,E1 125.311} C_DIS
LIN {X -0.113,Y -464.309,Z 239.486,A 0.000,B 0.000,C 90.000,E1 123.452} C_DIS
LIN {X 0.058,Y -462.224,Z 239.479,A 0.000,B 0.000,C 90.000,E1 122.163} C_DIS
LIN {X -0.076,Y -459.511,Z 239.470,A 0.000,B 0.000,C 90.000,E1 120.590} C_DIS
LIN {X 0.174,Y -457.331,Z 239.463,A 0.000,B 0.000,C 90.000,E1 119.283} C_DIS
LIN {X -0.022,Y -453.854,Z 239.452,A 0.000,B 0.000,C 90.000,E1 117.385} C_DIS
LIN {X -0.110,Y -450.366,Z 239.441,A 0.000,B 0.000,C 90.000,E1 115.463} C_DIS
LIN {X 0.151,Y -447.375,Z 239.432,A 0.000,B 0.000,C 90.000,E1 113.695} C_DIS
LIN {X 0.111,Y -447.385,Z 239.432,A 0.000,B 0.000,C 90.000,E1 113.695} C_DIS
LIN {X 0.105,Y -456.859,Z 239.411,A 0.000,B 0.000,C 90.000,E1 109.939} C_DIS
LIN {X 0.006,Y -457.589,Z 239.409,A 0.000,B 0.000,C 90.000,E1 109.631} C_DIS
LIN {X 0.093,Y -466.298,Z 239.386,A 0.000,B 0.000,C 90.000,E1 105.481} C_DIS
LIN {X 0.267,Y -467.845,Z 239.383,A 0.000,B 0.000,C 90.000,E1 104.828} C_DIS
LIN {X -0.171,Y -475.401,Z 239.358,A 0.000,B 0.000,C 90.000,E1 100.489} C_DIS
LIN {X 0.134,Y -476.054,Z 239.356,A 0.000,B 0.000,C 90.000,E1 100.141} C_DIS
LIN {X -0.061,Y -481.981,Z 239.331,A 0.000,B 0.000,C 90.000,E1 95.511} C_DIS
LIN {X 0.072,Y -482.356,Z 239.327,A 0.000,B 0.000,C 90.000,E1 94.878} C_DIS
LIN {X 0.209,Y -485.434,Z 239.305,A 0.000,B 0.000,C 90.000,E1 90.859} C_DIS
LIN {X -0.138,Y -485.505,Z 239.302,A 0.000,B 0.000,C 90.000,E1 90.286} C_DIS
LIN {X 0.242,Y -486.377,Z 239.281,A 0.000,B 0.000,C 90.000,E1 86.560} C_DIS
LIN {X 0.067,Y -486.366,Z 239.279,A 0.000,B 0.000,C 90.000,E1 86.274} C_DIS
LIN {X 0.155,Y -484.690,Z 239.254,A 0.000,B 0.000,C 90.000,E1 81.659} C_DIS
LIN {X -0.047,Y -484.456,Z 239.252,A 0.000,B 0.000,C 90.000,E1 81.376} C_DIS
LIN {X -0.043,Y -480.647,Z 239.228,A 0.000,B 0.000,C 90.000,E1 77.061} C_DIS
LIN {X -0.077,Y -480.369,Z 239.226,A 0.000,B 0.000,C 90.000,E1 76.756} C_DIS
LIN {X 0.147,Y -474.167,Z 239.201,A 0.000,B 0.000,C 90.000,E1 72.072} C_DIS
LIN {X 0.134,Y -469.473,Z 239.187,A 0.000,B 0.000,C 90.000,E1 69.571} C_DIS
LIN {X 0.159,Y -465.658,Z 239.173,A 0.000,B 0.000,C 90.000,E1 67.050} C_DIS
LIN {X -0.150,Y -462.733,Z 239.165,A 0.000,B 0.000,C 90.000,E1 65.793} C_DIS
LIN {X -0.189,Y -462.729,Z 239.165,A 0.000,B 0.000,C 90.000,E1 65.793} C_DIS
LIN {X 0.064,Y -467.475,Z 239.155,A 0.000,B 0.000,C 90.000,E1 63.896} C_DIS
LIN {X -0.236,Y -471.601,Z 239.146,A 0.000,B 0.000,C 90.000,E1 62.359} C_DIS
LIN {X -0.243,Y -475.710,Z 239.138,A 0.000,B 0.000,C 90.000,E1 60.795} C_DIS
LIN {X 0.065,Y -479.859,Z 239.129,A 0.000,B 0.000,C 90.000,E1 59.203} C_DIS
LIN {X 0.078,Y -485.779,Z 239.117,A 0.000,B 0.000,C 90.000,E1 57.041} C_DIS
LIN {X 0.026,Y -489.837,Z 239.108,A 0.000,B 0.000,C 90.000,E1 55.515} C_DIS
LIN {X 0.044,Y -493.492,Z 239.100,A 0.000,B 0.000,C 90.000,E1 53.989} C_DIS
LIN {X 0.001,Y -495.622,Z 239.095,A 0.000,B 0.000,C 90.000,E1 53.084} C_DIS
LIN {X -0.251,Y -498.119,Z 239.088,A 0.000,B 0.000,C 90.000,E1 51.904} C_DIS
LIN {X -0.073,Y -500.319,Z 239.082,A 0.000,B 0.000,C 90.000,E1 50.678} C_DIS
LIN {X 0.068,Y -502.279,Z 239.075,A 0.000,B 0.000,C 90.000,E1 49.461} C_DIS
LIN {X 0.031,Y -503.682,Z 239.070,A 0.000,B 0.000,C 90.000,E1 48.566} C_DIS
LIN {X -0.030,Y -504.911,Z 239.065,A 0.000,B 0.000,C 90.000,E1 47.676} C_DIS
LIN {X 0.182,Y -506.169,Z 239.058,A 0.000,B 0.000,C 90.000,E1 46.458} C_DIS
LIN {X 0.034,Y -507.129,Z 239.052,A 0.000,B 0.000,C 90.000,E1 45.283} C_DIS
LIN {X -0.102,Y -507.777,Z 239.045,A 0.000,B 0.000,C 90.000,E1 44.109} C_DIS
LIN {X -0.111,Y -508.091,Z 239.040,A 0.000,B 0.000,C 90.000,E1 43.218} C_DIS
LIN {X 0.146,Y -508.094,Z 239.033,A 0.000,B 0.000,C 90.000,E1 42.000} C_DIS
LIN {X -0.206,Y -507.974,Z 239.029,A 0.000,B 0.000,C 90.000,E1 41.148} C_DIS
LIN {X -0.050,Y -507.306,Z 239.020,A 0.000,B 0.000,C 90.000,E1 39.644} C_DIS
LIN {X -0.028,Y -506.795,Z 239.015,A 0.000,B 0.000,C 90.000,E1 38.749} C_DIS
LIN {X -0.120,Y -505.588,Z 239.009,A 0.000,B 0.000,C 90.000,E1 37.569} C_DIS
LIN {X -0.135,Y -504.089,Z 239.002,A 0.000,B 0.000,C 90.000,E1 36.377} C_DIS
LIN {X -0.276,Y -501.874,Z 238.994,A 0.000,B 0.000,C 90.000,E1 34.898} C_DIS
LIN {X -0.050,Y -499.298,Z 238.985,A 0.000,B 0.000,C 90.000,E1 33.372} C_DIS
LIN {X 0.256,Y -497.179,Z 238.979,A 0.000,B 0.000,C 90.000,E1 32.133} C_DIS
LIN {X -0.152,Y -492.511,Z 238.962,A 0.000,B 0.000,C 90.000,E1 29.155} C_DIS
LIN {X 0.206,Y -490.752,Z 238.955,A 0.000,B 0.000,C 90.000,E1 27.897} C_DIS
LIN {X -0.007,Y -487.083,Z 238.935,A 0.000,B 0.000,C 90.000,E1 24.259} C_DIS
LIN {X 0.098,Y -485.479,Z 238.925,A 0.000,B 0.000,C 90.000,E1 22.408} C_DIS
LIN {X 0.194,Y -483.355,Z 238.911,A 0.000,B 0.000,C 90.000,E1 19.939} C_DIS
LIN {X -0.123,Y -481.323,Z 238.897,A 0.000,B 0.000,C 90.000,E1 17.511} C_DIS
LIN {X -0.142,Y -480.215,Z 238.889,A 0.000,B 0.000,C 90.000,E1 15.969} C_DIS
LIN {X 0.087,Y -478.011,Z 238.870,A 0.000,B 0.000,C 90.000,E1 12.535} C_DIS
LIN {X -0.105,Y -476.843,Z 238.856,A 0.000,B 0.000,C 90.000,E1 10.074} C_DIS
LIN {X 0.119,Y -476.133,Z 238.844,A 0.000,B 0.000,C 90.000,E1 7.871} C_DIS
LIN {X 0.204,Y -475.674,Z 238.832,A 0.000,B 0.000,C 90.000,E1 5.682} C_DIS
LIN {X -0.152,Y -475.567,Z 238.816,A 0.000,B 0.000,C 90.000,E1 2.922} C_DIS
LIN {X 0.000,Y -476.147,Z 238.800,A 0.000,B 0.000,C 90.000,E1 360.000} C_DIS
LIN {X 0.084,Y -478.012,Z 238.782,A 0.000,B 0.000,C 90.000,E1 356.674} C_DIS
LIN {X 0.204,Y -479.630,Z 238.770,A 0.000,B 0.000,C 90.000,E1 354.489} C_DIS
LIN {X -0.013,Y -484.272,Z 238.747,A 0.000,B 0.000,C 90.000,E1 350.500} C_DIS
LIN {X -0.264,Y -487.083,Z 238.739,A 0.000,B 0.000,C 90.000,E1 348.993} C_DIS
LIN {X -0.018,Y -492.197,Z 238.727,A 0.000,B 0.000,C 90.000,E1 346.825} C_DIS
LIN {X 0.194,Y -496.340,Z 238.718,A 0.000,B 0.000,C 90.000,E1 345.283} C_DIS
LIN {X -0.074,Y -501.274,Z 238.708,A 0.000,B 0.000,C 90.000,E1 343.504} C_DIS
LIN {X -0.019,Y -507.095,Z 238.697,A 0.000,B 0.000,C 90.000,E1 341.402} C_DIS
LIN {X -0.122,Y -517.130,Z 238.679,A 0.000,B 0.000,C 90.000,E1 338.156} C_DIS
LIN {X 0.256,Y -523.171,Z 238.669,A 0.000,B 0.000,C 90.000,E1 336.357} C_DIS
LIN {X -0.199,Y -529.256,Z 238.659,A 0.000,B 0.000,C 90.000,E1 334.665} C_DIS
LIN {X -0.151,Y -537.705,Z 238.646,A 0.000,B 0.000,C 90.000,E1 332.359} C_DIS
LIN {X -0.308,Y -544.216,Z 238.637,A 0.000,B 0.000,C 90.000,E1 330.667} C_DIS
LIN {X -0.065,Y -547.376,Z 238.632,A 0.000,B 0.000,C 90.000,E1 329.793} C_DIS
LIN {X 0.312,Y -554.551,Z 238.621,A 0.000,B 0.000,C 90.000,E1 327.788} C_DIS
LIN {X -0.078,Y -561.824,Z 238.610,A 0.000,B 0.000,C 90.000,E1 325.881} C_DIS
LIN {X 0.110,Y -567.135,Z 238.603,A 0.000,B 0.000,C 90.000,E1 324.482} C_DIS
LIN {X -0.068,Y -572.227,Z 238.595,A 0.000,B 0.000,C 90.000,E1 323.130} C_DIS
LIN {X 0.191,Y -576.924,Z 238.588,A 0.000,B 0.000,C 90.000,E1 321.743} C_DIS
LIN {X 0.257,Y -587.725,Z 238.571,A 0.000,B 0.000,C 90.000,E1 318.771} C_DIS
LIN {X -0.108,Y -593.146,Z 238.564,A 0.000,B 0.000,C 90.000,E1 317.472} C_DIS
LIN {X 0.034,Y -596.315,Z 238.559,A 0.000,B 0.000,C 90.000,E1 316.662} C_DIS
LIN {X 0.012,Y -600.142,Z 238.553,A 0.000,B 0.000,C 90.000,E1 315.607} C_DIS
LIN {X 0.010,Y -601.930,Z 238.551,A 0.000,B 0.000,C 90.000,E1 315.081} C_DIS
LIN {X 0.049,Y -605.245,Z 238.545,A 0.000,B 0.000,C 90.000,E1 314.028} C_DIS
LIN {X 0.128,Y -607.897,Z 238.539,A 0.000,B 0.000,C 90.000,E1 312.975} C_DIS
LIN {X 0.274,Y -610.115,Z 238.533,A 0.000,B 0.000,C 90.000,E1 311.919} C_DIS
LIN {X -0.003,Y -611.786,Z 238.527,A 0.000,B 0.000,C 90.000,E1 310.906} C_DIS
LIN {X 0.200,Y -613.281,Z 238.522,A 0.000,B 0.000,C 90.000,E1 309.850} C_DIS
LIN {X -0.262,Y -614.276,Z 238.517,A 0.000,B 0.000,C 90.000,E1 309.116} C_DIS
LIN {X -0.112,Y -615.838,Z 238.510,A 0.000,B 0.000,C 90.000,E1 307.810} C_DIS
LIN {X -0.058,Y -616.600,Z 238.506,A 0.000,B 0.000,C 90.000,E1 307.030} C_DIS
LIN {X -0.180,Y -617.156,Z 238.500,A 0.000,B 0.000,C 90.000,E1 306.011} C_DIS
LIN {X 0.152,Y -617.633,Z 238.493,A 0.000,B 0.000,C 90.000,E1 304.692} C_DIS
LIN {X -0.020,Y -617.849,Z 238.486,A 0.000,B 0.000,C 90.000,E1 303.420} C_DIS
LIN {X -0.325,Y -617.429,Z 238.480,A 0.000,B 0.000,C 90.000,E1 302.418} C_DIS
LIN {X 0.221,Y -616.465,Z 238.474,A 0.000,B 0.000,C 90.000,E1 301.337} C_DIS
LIN {X -0.095,Y -614.944,Z 238.469,A 0.000,B 0.000,C 90.000,E1 300.335} C_DIS
LIN {X 0.130,Y -613.668,Z 238.464,A 0.000,B 0.000,C 90.000,E1 299.539} C_DIS
LIN {X 0.304,Y -611.493,Z 238.458,A 0.000,B 0.000,C 90.000,E1 298.487} C_DIS
LIN {X 0.161,Y -609.265,Z 238.453,A 0.000,B 0.000,C 90.000,E1 297.462} C_DIS
LIN {X -0.006,Y -606.602,Z 238.447,A 0.000,B 0.000,C 90.000,E1 296.437} C_DIS
LIN {X -0.266,Y -603.216,Z 238.440,A 0.000,B 0.000,C 90.000,E1 295.155} C_DIS
LIN {X 0.025,Y -600.395,Z 238.434,A 0.000,B 0.000,C 90.000,E1 294.079} C_DIS
LIN {X 0.051,Y -593.322,Z 238.418,A 0.000,B 0.000,C 90.000,E1 291.173} C_DIS
LIN {X 0.077,Y -589.766,Z 238.409,A 0.000,B 0.000,C 90.000,E1 289.577} C_DIS
LIN {X 0.239,Y -585.797,Z 238.398,A 0.000,B 0.000,C 90.000,E1 287.692} C_DIS
LIN {X 0.172,Y -581.530,Z 238.387,A 0.000,B 0.000,C 90.000,E1 285.552} C_DIS
LIN {X 0.209,Y -577.325,Z 238.373,A 0.000,B 0.000,C 90.000,E1 283.119} C_DIS
LIN {X -0.026,Y -572.468,Z 238.353,A 0.000,B 0.000,C 90.000,E1 279.613} C_DIS
LIN {X -0.267,Y -569.906,Z 238.340,A 0.000,B 0.000,C 90.000,E1 277.182} C_DIS
LIN {X 0.105,Y -567.402,Z 238.317,A 0.000,B 0.000,C 90.000,E1 273.037} C_DIS
LIN {X 0.054,Y -567.183,Z 238.303,A 0.000,B 0.000,C 90.000,E1 270.573} C_DIS
LIN {X -0.073,Y -568.309,Z 238.283,A 0.000,B 0.000,C 90.000,E1 267.020} C_DIS
LIN {X 0.169,Y -571.816,Z 238.262,A 0.000,B 0.000,C 90.000,E1 263.166} C_DIS
LIN {X 0.022,Y -573.780,Z 238.253,A 0.000,B 0.000,C 90.000,E1 261.546} C_DIS
LIN {X -0.088,Y -575.994,Z 238.244,A 0.000,B 0.000,C 90.000,E1 259.926} C_DIS
LIN {X 0.051,Y -578.454,Z 238.235,A 0.000,B 0.000,C 90.000,E1 258.285} C_DIS
LIN {X 0.249,Y -581.116,Z 238.226,A 0.000,B 0.000,C 90.000,E1 256.645} C_DIS
LIN {X 0.072,Y -583.534,Z 238.217,A 0.000,B 0.000,C 90.000,E1 255.046} C_DIS
LIN {X -0.296,Y -585.434,Z 238.210,A 0.000,B 0.000,C 90.000,E1 253.740} C_DIS
LIN {X 0.010,Y -586.362,Z 238.205,A 0.000,B 0.000,C 90.000,E1 252.906} C_DIS
LIN {X -0.236,Y -587.018,Z 238.201,A 0.000,B 0.000,C 90.000,E1 252.127} C_DIS
LIN {X -0.150,Y -587.296,Z 238.198,A 0.000,B 0.000,C 90.000,E1 251.583} C_DIS
LIN {X 0.026,Y -587.562,Z 238.192,A 0.000,B 0.000,C 90.000,E1 250.496} C_DIS
LIN {X -0.017,Y -587.599,Z 238.187,A 0.000,B 0.000,C 90.000,E1 249.699} C_DIS
LIN {X -0.181,Y -587.430,Z 238.181,A 0.000,B 0.000,C 90.000,E1 248.646} C_DIS
LIN {X 0.200,Y -586.615,Z 238.175,A 0.000,B 0.000,C 90.000,E1 247.539} C_DIS
LIN {X 0.146,Y -585.785,Z 238.171,A 0.000,B 0.000,C 90.000,E1 246.741} C_DIS
LIN {X 0.313,Y -584.770,Z 238.166,A 0.000,B 0.000,C 90.000,E1 245.921} C_DIS
LIN {X 0.344,Y -582.881,Z 238.160,A 0.000,B 0.000,C 90.000,E1 244.845} C_DIS
LIN {X 0.088,Y -581.755,Z 238.158,A 0.000,B 0.000,C 90.000,E1 244.332} C_DIS
LIN {X 0.214,Y -579.912,Z 238.153,A 0.000,B 0.000,C 90.000,E1 243.512} C_DIS
LIN {X -0.201,Y -578.078,Z 238.149,A 0.000,B 0.000,C 90.000,E1 242.743} C_DIS
LIN {X -0.006,Y -575.239,Z 238.143,A 0.000,B 0.000,C 90.000,E1 241.641} C_DIS
LIN {X -0.193,Y -572.981,Z 238.138,A 0.000,B 0.000,C 90.000,E1 240.845} C_DIS
LIN {X -0.074,Y -569.824,Z 238.132,A 0.000,B 0.000,C 90.000,E1 239.744} C_DIS
LIN {X -0.209,Y -566.502,Z 238.126,A 0.000,B 0.000,C 90.000,E1 238.663} C_DIS
LIN {X 0.293,Y -563.930,Z 238.121,A 0.000,B 0.000,C 90.000,E1 237.788} C_DIS
LIN {X 0.077,Y -560.390,Z 238.115,A 0.000,B 0.000,C 90.000,E1 236.707} C_DIS
LIN {X -0.035,Y -555.195,Z 238.106,A 0.000,B 0.000,C 90.000,E1 235.055} C_DIS
LIN {X 0.253,Y -551.677,Z 238.100,A 0.000,B 0.000,C 90.000,E1 233.909} C_DIS
LIN {X -0.087,Y -544.573,Z 238.087,A 0.000,B 0.000,C 90.000,E1 231.698} C_DIS
LIN {X 0.007,Y -539.207,Z 238.078,A 0.000,B 0.000,C 90.000,E1 229.989} C_DIS
LIN {X 0.332,Y -533.790,Z 238.068,A 0.000,B 0.000,C 90.000,E1 228.243} C_DIS
LIN {X 0.249,Y -530.912,Z 238.063,A 0.000,B 0.000,C 90.000,E1 227.391} C_DIS
LIN {X 0.168,Y -529.153,Z 238.060,A 0.000,B 0.000,C 90.000,E1 226.824} C_DIS
LIN {X 0.239,Y -523.464,Z 238.051,A 0.000,B 0.000,C 90.000,E1 225.081} C_DIS
LIN {X -0.034,Y -519.791,Z 238.044,A 0.000,B 0.000,C 90.000,E1 223.947} C_DIS
LIN {X -0.250,Y -513.324,Z 238.033,A 0.000,B 0.000,C 90.000,E1 221.919} C_DIS
LIN {X 0.174,Y -510.678,Z 238.028,A 0.000,B 0.000,C 90.000,E1 220.987} C_DIS
LIN {X 0.157,Y -504.505,Z 238.016,A 0.000,B 0.000,C 90.000,E1 218.910} C_DIS
LIN {X -0.204,Y -499.450,Z 238.006,A 0.000,B 0.000,C 90.000,E1 217.156} C_DIS
LIN {X 0.116,Y -494.386,Z 237.996,A 0.000,B 0.000,C 90.000,E1 215.311} C_DIS
LIN {X 0.190,Y -490.060,Z 237.988,A 0.000,B 0.000,C 90.000,E1 213.785} C_DIS
LIN {X -0.057,Y -486.741,Z 237.981,A 0.000,B 0.000,C 90.000,E1 212.594} C_DIS
LIN {X 0.002,Y -480.063,Z 237.967,A 0.000,B 0.000,C 90.000,E1 210.129} C_DIS
LIN {X 0.140,Y -471.800,Z 237.948,A 0.000,B 0.000,C 90.000,E1 206.693} C_DIS
LIN {X -0.064,Y -466.645,Z 237.934,A 0.000,B 0.000,C 90.000,E1 204.207} C_DIS
LIN {X -0.176,Y -460.322,Z 237.915,A 0.000,B 0.000,C 90.000,E1 200.737} C_DIS
LIN {X -0.058,Y -456.804,Z 237.903,A 0.000,B 0.000,C 90.000,E1 198.489} C_DIS
LIN {X 0.057,Y -454.120,Z 237.892,A 0.000,B 0.000,C 90.000,E1 196.551} C_DIS
LIN {X 0.088,Y -450.354,Z 237.876,A 0.000,B 0.000,C 90.000,E1 193.647} C_DIS
LIN {X -0.240,Y -447.568,Z 237.863,A 0.000,B 0.000,C 90.000,E1 191.422} C_DIS
LIN {X -0.018,Y -445.347,Z 237.852,A 0.000,B 0.000,C 90.000,E1 189.443} C_DIS
LIN {X -0.026,Y -442.632,Z 237.838,A 0.000,B 0.000,C 90.000,E1 186.834} C_DIS
LIN {X -0.098,Y -440.870,Z 237.827,A 0.000,B 0.000,C 90.000,E1 184.878} C_DIS
LIN {X -0.212,Y -439.314,Z 237.816,A 0.000,B 0.000,C 90.000,E1 182.922} C_DIS
LIN {X 0.132,Y -437.564,Z 237.803,A 0.000,B 0.000,C 90.000,E1 180.573} C_DIS
LIN {X 0.098,Y -436.008,Z 237.789,A 0.000,B 0.000,C 90.000,E1 177.936} C_DIS
LIN {X 0.031,Y -435.150,Z 237.774,A 0.000,B 0.000,C 90.000,E1 175.298} C_DIS
LIN {X -0.164,Y -434.963,Z 237.763,A 0.000,B 0.000,C 90.000,E1 173.337} C_DIS
LIN {X -0.100,Y -435.203,Z 237.748,A 0.000,B 0.000,C 90.000,E1 170.679} C_DIS
LIN {X -0.110,Y -435.871,Z 237.732,A 0.000,B 0.000,C 90.000,E1 167.701} C_DIS
LIN {X -0.034,Y -437.014,Z 237.717,A 0.000,B 0.000,C 90.000,E1 165.046} C_DIS
LIN {X 0.107,Y -437.892,Z 237.708,A 0.000,B 0.000,C 90.000,E1 163.378} C_DIS
LIN {X -0.158,Y -438.776,Z 237.699,A 0.000,B 0.000,C 90.000,E1 161.764} C_DIS
LIN {X 0.127,Y -440.123,Z 237.688,A 0.000,B 0.000,C 90.000,E1 159.752} C_DIS
LIN {X 0.168,Y -442.707,Z 237.671,A 0.000,B 0.000,C 90.000,E1 156.794} C_DIS
LIN {X -0.072,Y -445.213,Z 237.659,A 0.000,B 0.000,C 90.000,E1 154.537} C_DIS
LIN {X 0.211,Y -447.136,Z 237.649,A 0.000,B 0.000,C 90.000,E1 152.871} C_DIS
LIN {X 0.204,Y -448.485,Z 237.644,A 0.000,B 0.000,C 90.000,E1 151.897} C_DIS
LIN {X -0.072,Y -451.884,Z 237.631,A 0.000,B 0.000,C 90.000,E1 149.665} C_DIS
LIN {X 0.105,Y -454.984,Z 237.621,A 0.000,B 0.000,C 90.000,E1 147.709} C_DIS
LIN {X -0.190,Y -459.187,Z 237.606,A 0.000,B 0.000,C 90.000,E1 145.182} C_DIS
LIN {X -0.220,Y -461.366,Z 237.599,A 0.000,B 0.000,C 90.000,E1 143.909} C_DIS
LIN {X -0.069,Y -464.339,Z 237.589,A 0.000,B 0.000,C 90.000,E1 141.984} C_DIS
LIN {X 0.307,Y -466.508,Z 237.580,A 0.000,B 0.000,C 90.000,E1 140.356} C_DIS
LIN {X -0.290,Y -468.379,Z 237.571,A 0.000,B 0.000,C 90.000,E1 138.852} C_DIS
LIN {X 0.040,Y -469.684,Z 237.564,A 0.000,B 0.000,C 90.000,E1 137.553} C_DIS
LIN {X -0.042,Y -470.447,Z 237.559,A 0.000,B 0.000,C 90.000,E1 136.620} C_DIS
LIN {X -0.034,Y -471.097,Z 237.552,A 0.000,B 0.000,C 90.000,E1 135.364} C_DIS
LIN {X -0.018,Y -471.521,Z 237.545,A 0.000,B 0.000,C 90.000,E1 134.109} C_DIS
LIN {X -0.076,Y -471.617,Z 237.540,A 0.000,B 0.000,C 90.000,E1 133.176} C_DIS
LIN {X -0.131,Y -471.443,Z 237.535,A 0.000,B 0.000,C 90.000,E1 132.243} C_DIS
LIN {X -0.107,Y -470.736,Z 237.528,A 0.000,B 0.000,C 90.000,E1 130.987} C_DIS
LIN {X -0.051,Y -469.978,Z 237.521,A 0.000,B 0.000,C 90.000,E1 129.725} C_DIS
LIN {X -0.003,Y -469.033,Z 237.514,A 0.000,B 0.000,C 90.000,E1 128.463} C_DIS
LIN {X 0.161,Y -467.502,Z 237.505,A 0.000,B 0.000,C 90.000,E1 126.870} C_DIS
LIN {X -0.127,Y -465.936,Z 237.498,A 0.000,B 0.000,C 90.000,E1 125.644} C_DIS
LIN {X -0.086,Y -464.609,Z 237.493,A 0.000,B 0.000,C 90.000,E1 124.692} C_DIS
LIN {X 0.087,Y -462.200,Z 237.484,A 0.000,B 0.000,C 90.000,E1 123.086} C_DIS
LIN {X 0.218,Y -460.094,Z 237.477,A 0.000,B 0.000,C 90.000,E1 121.799} C_DIS
LIN {X -0.086,Y -456.837,Z 237.466,A 0.000,B 0.000,C 90.000,E1 119.922} C_DIS
LIN {X 0.120,Y -454.577,Z 237.459,A 0.000,B 0.000,C 90.000,E1 118.615} C_DIS
LIN {X 0.050,Y -451.065,Z 237.448,A 0.000,B 0.000,C 90.000,E1 116.693} C_DIS
LIN {X 0.237,Y -446.522,Z 237.434,A 0.000,B 0.000,C 90.000,E1 114.079} C_DIS
LIN {X 0.197,Y -446.524,Z 237.434,A 0.000,B 0.000,C 90.000,E1 114.079} C_DIS
LIN {X -0.065,Y -455.197,Z 237.414,A 0.000,B 0.000,C 90.000,E1 110.556} C_DIS
LIN {X 0.161,Y -456.992,Z 237.411,A 0.000,B 0.000,C 90.000,E1 109.885} C_DIS
LIN {X -0.031,Y -458.251,Z 237.407,A 0.000,B 0.000,C 90.000,E1 109.268} C_DIS
LIN {X 0.167,Y -466.412,Z 237.386,A 0.000,B 0.000,C 90.000,E1 105.426} C_DIS
LIN {X -0.109,Y -467.921,Z 237.382,A 0.000,B 0.000,C 90.000,E1 104.828} C_DIS
LIN {X -0.082,Y -475.495,Z 237.358,A 0.000,B 0.000,C 90.000,E1 100.433} C_DIS
LIN {X -0.244,Y -476.136,Z 237.356,A 0.000,B 0.000,C 90.000,E1 100.141} C_DIS
LIN {X 0.040,Y -482.051,Z 237.330,A 0.000,B 0.000,C 90.000,E1 95.454} C_DIS
LIN {X -0.170,Y -485.481,Z 237.305,A 0.000,B 0.000,C 90.000,E1 90.859} C_DIS
LIN {X -0.138,Y -486.386,Z 237.281,A 0.000,B 0.000,C 90.000,E1 86.560} C_DIS
LIN {X 0.173,Y -486.363,Z 237.279,A 0.000,B 0.000,C 90.000,E1 86.216} C_DIS
LIN {X 0.255,Y -484.689,Z 237.254,A 0.000,B 0.000,C 90.000,E1 81.602} C_DIS
LIN {X 0.135,Y -483.353,Z 237.247,A 0.000,B 0.000,C 90.000,E1 80.387} C_DIS
LIN {X 0.155,Y -480.623,Z 237.228,A 0.000,B 0.000,C 90.000,E1 76.992} C_DIS
LIN {X 0.012,Y -480.292,Z 237.226,A 0.000,B 0.000,C 90.000,E1 76.700} C_DIS
LIN {X -0.083,Y -474.114,Z 237.200,A 0.000,B 0.000,C 90.000,E1 72.054} C_DIS
LIN {X -0.215,Y -465.574,Z 237.172,A 0.000,B 0.000,C 90.000,E1 67.050} C_DIS
LIN {X 0.218,Y -462.004,Z 237.164,A 0.000,B 0.000,C 90.000,E1 65.409} C_DIS
LIN {X 0.178,Y -462.008,Z 237.164,A 0.000,B 0.000,C 90.000,E1 65.409} C_DIS
LIN {X 0.150,Y -467.698,Z 237.151,A 0.000,B 0.000,C 90.000,E1 63.204} C_DIS
LIN {X -0.233,Y -473.471,Z 237.139,A 0.000,B 0.000,C 90.000,E1 61.051} C_DIS
LIN {X -0.018,Y -478.402,Z 237.129,A 0.000,B 0.000,C 90.000,E1 59.154} C_DIS
LIN {X -0.054,Y -484.321,Z 237.117,A 0.000,B 0.000,C 90.000,E1 56.993} C_DIS
LIN {X -0.143,Y -488.380,Z 237.108,A 0.000,B 0.000,C 90.000,E1 55.468} C_DIS
LIN {X 0.129,Y -491.990,Z 237.100,A 0.000,B 0.000,C 90.000,E1 53.909} C_DIS
LIN {X 0.070,Y -494.089,Z 237.095,A 0.000,B 0.000,C 90.000,E1 53.004} C_DIS
LIN {X -0.062,Y -495.967,Z 237.090,A 0.000,B 0.000,C 90.000,E1 52.110} C_DIS
LIN {X 0.088,Y -498.244,Z 237.083,A 0.000,B 0.000,C 90.000,E1 50.884} C_DIS
LIN {X -0.057,Y -501.089,Z 237.073,A 0.000,B 0.000,C 90.000,E1 49.094} C_DIS
LIN {X 0.097,Y -502.775,Z 237.066,A 0.000,B 0.000,C 90.000,E1 47.877} C_DIS
LIN {X -0.097,Y -504.143,Z 237.059,A 0.000,B 0.000,C 90.000,E1 46.701} C_DIS
LIN {X 0.079,Y -505.142,Z 237.053,A 0.000,B 0.000,C 90.000,E1 45.486} C_DIS
LIN {X 0.274,Y -505.799,Z 237.046,A 0.000,B 0.000,C 90.000,E1 44.271} C_DIS
LIN {X -0.103,Y -506.119,Z 237.041,A 0.000,B 0.000,C 90.000,E1 43.419} C_DIS
LIN {X -0.130,Y -506.211,Z 237.036,A 0.000,B 0.000,C 90.000,E1 42.528} C_DIS
LIN {X 0.102,Y -506.024,Z 237.030,A 0.000,B 0.000,C 90.000,E1 41.310} C_DIS
LIN {X 0.111,Y -505.729,Z 237.025,A 0.000,B 0.000,C 90.000,E1 40.415} C_DIS
LIN {X -0.270,Y -505.268,Z 237.020,A 0.000,B 0.000,C 90.000,E1 39.564} C_DIS
LIN {X 0.122,Y -504.614,Z 237.015,A 0.000,B 0.000,C 90.000,E1 38.624} C_DIS
LIN {X 0.002,Y -503.389,Z 237.008,A 0.000,B 0.000,C 90.000,E1 37.443} C_DIS
LIN {X 0.139,Y -501.386,Z 237.000,A 0.000,B 0.000,C 90.000,E1 35.931} C_DIS
LIN {X -0.099,Y -500.449,Z 236.996,A 0.000,B 0.000,C 90.000,E1 35.358} C_DIS
LIN {X 0.092,Y -497.918,Z 236.988,A 0.000,B 0.000,C 90.000,E1 33.833} C_DIS
LIN {X 0.235,Y -494.668,Z 236.978,A 0.000,B 0.000,C 90.000,E1 32.005} C_DIS
LIN {X 0.205,Y -492.681,Z 236.971,A 0.000,B 0.000,C 90.000,E1 30.797} C_DIS
LIN {X 0.155,Y -490.408,Z 236.963,A 0.000,B 0.000,C 90.000,E1 29.283} C_DIS
LIN {X -0.114,Y -487.201,Z 236.949,A 0.000,B 0.000,C 90.000,E1 26.873} C_DIS
LIN {X 0.181,Y -484.745,Z 236.934,A 0.000,B 0.000,C 90.000,E1 24.079} C_DIS
LIN {X -0.026,Y -483.147,Z 236.924,A 0.000,B 0.000,C 90.000,E1 22.259} C_DIS
LIN {X -0.187,Y -482.123,Z 236.917,A 0.000,B 0.000,C 90.000,E1 21.046} C_DIS
LIN {X 0.092,Y -480.322,Z 236.905,A 0.000,B 0.000,C 90.000,E1 18.852} C_DIS
LIN {X 0.162,Y -478.655,Z 236.893,A 0.000,B 0.000,C 90.000,E1 16.677} C_DIS
LIN {X 0.097,Y -477.574,Z 236.884,A 0.000,B 0.000,C 90.000,E1 15.134} C_DIS
LIN {X -0.206,Y -475.708,Z 236.867,A 0.000,B 0.000,C 90.000,E1 12.063} C_DIS
LIN {X -0.231,Y -474.904,Z 236.857,A 0.000,B 0.000,C 90.000,E1 10.197} C_DIS
LIN {X -0.048,Y -474.142,Z 236.844,A 0.000,B 0.000,C 90.000,E1 7.992} C_DIS
LIN {X 0.045,Y -473.676,Z 236.832,A 0.000,B 0.000,C 90.000,E1 5.796} C_DIS
LIN {X 0.092,Y -473.600,Z 236.817,A 0.000,B 0.000,C 90.000,E1 2.980} C_DIS
LIN {X -0.032,Y -474.424,Z 236.797,A 0.000,B 0.000,C 90.000,E1 359.484} C_DIS
LIN {X -0.201,Y -476.251,Z 236.780,A 0.000,B 0.000,C 90.000,E1 356.388} C_DIS
LIN {X -0.137,Y -477.925,Z 236.768,A 0.000,B 0.000,C 90.000,E1 354.204} C_DIS
LIN {X 0.044,Y -481.398,Z 236.751,A 0.000,B 0.000,C 90.000,E1 351.084} C_DIS
LIN {X -0.039,Y -483.298,Z 236.744,A 0.000,B 0.000,C 90.000,E1 349.859} C_DIS
LIN {X 0.017,Y -487.909,Z 236.732,A 0.000,B 0.000,C 90.000,E1 347.701} C_DIS
LIN {X -0.167,Y -494.390,Z 236.718,A 0.000,B 0.000,C 90.000,E1 345.283} C_DIS
LIN {X -0.004,Y -499.295,Z 236.708,A 0.000,B 0.000,C 90.000,E1 343.449} C_DIS
LIN {X 0.156,Y -505.094,Z 236.696,A 0.000,B 0.000,C 90.000,E1 341.329} C_DIS
LIN {X 0.159,Y -514.164,Z 236.680,A 0.000,B 0.000,C 90.000,E1 338.358} C_DIS
LIN {X 0.127,Y -521.170,Z 236.668,A 0.000,B 0.000,C 90.000,E1 336.305} C_DIS
LIN {X 0.160,Y -526.286,Z 236.660,A 0.000,B 0.000,C 90.000,E1 334.845} C_DIS
LIN {X 0.134,Y -534.766,Z 236.648,A 0.000,B 0.000,C 90.000,E1 332.538} C_DIS
LIN {X -0.074,Y -541.225,Z 236.638,A 0.000,B 0.000,C 90.000,E1 330.845} C_DIS
LIN {X -0.130,Y -544.428,Z 236.633,A 0.000,B 0.000,C 90.000,E1 329.999} C_DIS
LIN {X 0.166,Y -551.685,Z 236.622,A 0.000,B 0.000,C 90.000,E1 327.995} C_DIS
LIN {X -0.215,Y -560.026,Z 236.610,A 0.000,B 0.000,C 90.000,E1 325.801} C_DIS
LIN {X -0.161,Y -564.287,Z 236.604,A 0.000,B 0.000,C 90.000,E1 324.689} C_DIS
LIN {X 0.067,Y -569.445,Z 236.596,A 0.000,B 0.000,C 90.000,E1 323.290} C_DIS
LIN {X 0.133,Y -573.346,Z 236.590,A 0.000,B 0.000,C 90.000,E1 322.190} C_DIS
LIN {X -0.035,Y -578.077,Z 236.583,A 0.000,B 0.000,C 90.000,E1 320.848} C_DIS
LIN {X 0.009,Y -591.705,Z 236.563,A 0.000,B 0.000,C 90.000,E1 317.349} C_DIS
LIN {X 0.132,Y -594.867,Z 236.559,A 0.000,B 0.000,C 90.000,E1 316.539} C_DIS
LIN {X 0.074,Y -598.715,Z 236.553,A 0.000,B 0.000,C 90.000,E1 315.486} C_DIS
LIN {X 0.072,Y -602.108,Z 236.547,A 0.000,B 0.000,C 90.000,E1 314.433} C_DIS
LIN {X -0.340,Y -603.630,Z 236.544,A 0.000,B 0.000,C 90.000,E1 313.947} C_DIS
LIN {X -0.088,Y -605.715,Z 236.540,A 0.000,B 0.000,C 90.000,E1 313.137} C_DIS
LIN {X 0.027,Y -607.899,Z 236.534,A 0.000,B 0.000,C 90.000,E1 312.081} C_DIS
LIN {X -0.277,Y -609.667,Z 236.528,A 0.000,B 0.000,C 90.000,E1 311.067} C_DIS
LIN {X -0.102,Y -611.168,Z 236.522,A 0.000,B 0.000,C 90.000,E1 310.011} C_DIS
LIN {X 0.279,Y -612.149,Z 236.518,A 0.000,B 0.000,C 90.000,E1 309.197} C_DIS
LIN {X 0.206,Y -613.896,Z 236.509,A 0.000,B 0.000,C 90.000,E1 307.649} C_DIS
LIN {X -0.060,Y -614.441,Z 236.506,A 0.000,B 0.000,C 90.000,E1 307.156} C_DIS
LIN {X 0.281,Y -615.029,Z 236.501,A 0.000,B 0.000,C 90.000,E1 306.091} C_DIS
LIN {X 0.074,Y -615.490,Z 236.494,A 0.000,B 0.000,C 90.000,E1 304.818} C_DIS
LIN {X 0.375,Y -615.747,Z 236.486,A 0.000,B 0.000,C 90.000,E1 303.499} C_DIS
LIN {X 0.081,Y -615.544,Z 236.482,A 0.000,B 0.000,C 90.000,E1 302.752} C_DIS
LIN {X -0.214,Y -615.040,Z 236.478,A 0.000,B 0.000,C 90.000,E1 302.005} C_DIS
LIN {X 0.011,Y -614.132,Z 236.473,A 0.000,B 0.000,C 90.000,E1 301.209} C_DIS
LIN {X -0.300,Y -613.078,Z 236.469,A 0.000,B 0.000,C 90.000,E1 300.463} C_DIS
LIN {X -0.166,Y -610.816,Z 236.462,A 0.000,B 0.000,C 90.000,E1 299.155} C_DIS
LIN {X -0.070,Y -608.065,Z 236.455,A 0.000,B 0.000,C 90.000,E1 297.847} C_DIS
LIN {X 0.070,Y -606.262,Z 236.450,A 0.000,B 0.000,C 90.000,E1 297.052} C_DIS
LIN {X 0.338,Y -602.907,Z 236.443,A 0.000,B 0.000,C 90.000,E1 295.720} C_DIS
LIN {X -0.246,Y -599.496,Z 236.436,A 0.000,B 0.000,C 90.000,E1 294.463} C_DIS
LIN {X -0.133,Y -591.687,Z 236.418,A 0.000,B 0.000,C 90.000,E1 291.280} C_DIS
LIN {X 0.078,Y -587.590,Z 236.408,A 0.000,B 0.000,C 90.000,E1 289.396} C_DIS
LIN {X 0.186,Y -583.653,Z 236.397,A 0.000,B 0.000,C 90.000,E1 287.511} C_DIS
LIN {X -0.159,Y -579.916,Z 236.387,A 0.000,B 0.000,C 90.000,E1 285.662} C_DIS
LIN {X -0.182,Y -575.701,Z 236.373,A 0.000,B 0.000,C 90.000,E1 283.231} C_DIS
LIN {X 0.059,Y -570.795,Z 236.354,A 0.000,B 0.000,C 90.000,E1 279.670} C_DIS
LIN {X 0.150,Y -568.436,Z 236.342,A 0.000,B 0.000,C 90.000,E1 277.473} C_DIS
LIN {X 0.048,Y -565.451,Z 236.310,A 0.000,B 0.000,C 90.000,E1 271.718} C_DIS
LIN {X 0.062,Y -566.225,Z 236.287,A 0.000,B 0.000,C 90.000,E1 267.593} C_DIS
LIN {X 0.160,Y -570.632,Z 236.259,A 0.000,B 0.000,C 90.000,E1 262.648} C_DIS
LIN {X 0.006,Y -573.774,Z 236.246,A 0.000,B 0.000,C 90.000,E1 260.208} C_DIS
LIN {X 0.207,Y -576.596,Z 236.235,A 0.000,B 0.000,C 90.000,E1 258.285} C_DIS
LIN {X -0.197,Y -579.291,Z 236.226,A 0.000,B 0.000,C 90.000,E1 256.700} C_DIS
LIN {X -0.186,Y -582.095,Z 236.216,A 0.000,B 0.000,C 90.000,E1 254.810} C_DIS
LIN {X -0.022,Y -583.935,Z 236.208,A 0.000,B 0.000,C 90.000,E1 253.449} C_DIS
LIN {X -0.119,Y -584.796,Z 236.204,A 0.000,B 0.000,C 90.000,E1 252.653} C_DIS
LIN {X 0.180,Y -585.405,Z 236.199,A 0.000,B 0.000,C 90.000,E1 251.819} C_DIS
LIN {X -0.219,Y -585.731,Z 236.193,A 0.000,B 0.000,C 90.000,E1 250.786} C_DIS
LIN {X -0.063,Y -585.816,Z 236.187,A 0.000,B 0.000,C 90.000,E1 249.699} C_DIS
LIN {X 0.294,Y -585.615,Z 236.181,A 0.000,B 0.000,C 90.000,E1 248.592} C_DIS
LIN {X 0.104,Y -584.801,Z 236.175,A 0.000,B 0.000,C 90.000,E1 247.539} C_DIS
LIN {X -0.097,Y -583.637,Z 236.169,A 0.000,B 0.000,C 90.000,E1 246.485} C_DIS
LIN {X 0.049,Y -582.441,Z 236.165,A 0.000,B 0.000,C 90.000,E1 245.665} C_DIS
LIN {X 0.317,Y -581.570,Z 236.162,A 0.000,B 0.000,C 90.000,E1 245.101} C_DIS
LIN {X 0.303,Y -579.250,Z 236.156,A 0.000,B 0.000,C 90.000,E1 244.024} C_DIS
LIN {X -0.264,Y -576.724,Z 236.150,A 0.000,B 0.000,C 90.000,E1 242.999} C_DIS
LIN {X -0.085,Y -573.975,Z 236.144,A 0.000,B 0.000,C 90.000,E1 241.897} C_DIS
LIN {X 0.215,Y -571.744,Z 236.139,A 0.000,B 0.000,C 90.000,E1 241.051} C_DIS
LIN {X -0.071,Y -567.776,Z 236.132,A 0.000,B 0.000,C 90.000,E1 239.715} C_DIS
LIN {X -0.036,Y -564.439,Z 236.126,A 0.000,B 0.000,C 90.000,E1 238.614} C_DIS
LIN {X -0.153,Y -560.136,Z 236.118,A 0.000,B 0.000,C 90.000,E1 237.248} C_DIS
LIN {X -0.340,Y -555.852,Z 236.110,A 0.000,B 0.000,C 90.000,E1 235.881} C_DIS
LIN {X -0.293,Y -551.381,Z 236.103,A 0.000,B 0.000,C 90.000,E1 234.482} C_DIS
LIN {X 0.046,Y -546.048,Z 236.093,A 0.000,B 0.000,C 90.000,E1 232.763} C_DIS
LIN {X -0.190,Y -541.633,Z 236.085,A 0.000,B 0.000,C 90.000,E1 231.376} C_DIS
LIN {X -0.103,Y -538.020,Z 236.079,A 0.000,B 0.000,C 90.000,E1 230.231} C_DIS
LIN {X -0.146,Y -534.382,Z 236.073,A 0.000,B 0.000,C 90.000,E1 229.094} C_DIS
LIN {X 0.116,Y -530.650,Z 236.066,A 0.000,B 0.000,C 90.000,E1 227.919} C_DIS
LIN {X -0.033,Y -526.993,Z 236.060,A 0.000,B 0.000,C 90.000,E1 226.782} C_DIS
LIN {X -0.019,Y -521.298,Z 236.050,A 0.000,B 0.000,C 90.000,E1 225.040} C_DIS
LIN {X -0.030,Y -516.656,Z 236.042,A 0.000,B 0.000,C 90.000,E1 223.581} C_DIS
LIN {X -0.141,Y -512.057,Z 236.034,A 0.000,B 0.000,C 90.000,E1 222.123} C_DIS
LIN {X 0.201,Y -505.762,Z 236.022,A 0.000,B 0.000,C 90.000,E1 220.011} C_DIS
LIN {X -0.020,Y -501.447,Z 236.014,A 0.000,B 0.000,C 90.000,E1 218.543} C_DIS
LIN {X -0.049,Y -496.412,Z 236.004,A 0.000,B 0.000,C 90.000,E1 216.744} C_DIS
LIN {X -0.049,Y -492.167,Z 235.996,A 0.000,B 0.000,C 90.000,E1 215.231} C_DIS
LIN {X 0.145,Y -488.728,Z 235.989,A 0.000,B 0.000,C 90.000,E1 213.992} C_DIS
LIN {X 0.110,Y -484.512,Z 235.980,A 0.000,B 0.000,C 90.000,E1 212.467} C_DIS
LIN {X 0.103,Y -477.799,Z 235.967,A 0.000,B 0.000,C 90.000,E1 210.001} C_DIS
LIN {X -0.168,Y -468.250,Z 235.944,A 0.000,B 0.000,C 90.000,E1 205.976} C_DIS
LIN {X -0.187,Y -463.826,Z 235.932,A 0.000,B 0.000,C 90.000,E1 203.770} C_DIS
LIN {X 0.101,Y -458.200,Z 235.914,A 0.000,B 0.000,C 90.000,E1 200.556} C_DIS
LIN {X 0.054,Y -454.231,Z 235.900,A 0.000,B 0.000,C 90.000,E1 198.000} C_DIS
LIN {X 0.094,Y -452.038,Z 235.891,A 0.000,B 0.000,C 90.000,E1 196.386} C_DIS
LIN {X -0.113,Y -448.699,Z 235.877,A 0.000,B 0.000,C 90.000,E1 193.828} C_DIS
LIN {X 0.048,Y -445.888,Z 235.864,A 0.000,B 0.000,C 90.000,E1 191.535} C_DIS
LIN {X -0.215,Y -443.656,Z 235.853,A 0.000,B 0.000,C 90.000,E1 189.613} C_DIS
LIN {X 0.154,Y -440.892,Z 235.839,A 0.000,B 0.000,C 90.000,E1 186.947} C_DIS
LIN {X 0.038,Y -439.098,Z 235.828,A 0.000,B 0.000,C 90.000,E1 184.992} C_DIS
LIN {X 0.189,Y -437.797,Z 235.819,A 0.000,B 0.000,C 90.000,E1 183.326} C_DIS
LIN {X 0.072,Y -436.013,Z 235.806,A 0.000,B 0.000,C 90.000,E1 181.031} C_DIS
LIN {X -0.024,Y -434.352,Z 235.791,A 0.000,B 0.000,C 90.000,E1 178.396} C_DIS
LIN {X -0.039,Y -433.289,Z 235.775,A 0.000,B 0.000,C 90.000,E1 175.412} C_DIS
LIN {X 0.154,Y -433.090,Z 235.763,A 0.000,B 0.000,C 90.000,E1 173.394} C_DIS
LIN {X 0.163,Y -433.341,Z 235.749,A 0.000,B 0.000,C 90.000,E1 170.735} C_DIS
LIN {X 0.214,Y -434.101,Z 235.730,A 0.000,B 0.000,C 90.000,E1 167.409} C_DIS
LIN {X -0.189,Y -435.272,Z 235.716,A 0.000,B 0.000,C 90.000,E1 164.810} C_DIS
LIN {X -0.084,Y -436.172,Z 235.706,A 0.000,B 0.000,C 90.000,E1 163.142} C_DIS
LIN {X 0.165,Y -437.065,Z 235.697,A 0.000,B 0.000,C 90.000,E1 161.456} C_DIS
LIN {X 0.100,Y -438.745,Z 235.684,A 0.000,B 0.000,C 90.000,E1 159.156} C_DIS
LIN {X -0.156,Y -441.450,Z 235.668,A 0.000,B 0.000,C 90.000,E1 156.230} C_DIS
LIN {X 0.114,Y -443.649,Z 235.657,A 0.000,B 0.000,C 90.000,E1 154.229} C_DIS
LIN {X -0.060,Y -446.990,Z 235.642,A 0.000,B 0.000,C 90.000,E1 151.641} C_DIS
LIN {X 0.156,Y -449.959,Z 235.632,A 0.000,B 0.000,C 90.000,E1 149.665} C_DIS
LIN {X -0.245,Y -453.526,Z 235.619,A 0.000,B 0.000,C 90.000,E1 147.454} C_DIS
LIN {X 0.109,Y -456.155,Z 235.610,A 0.000,B 0.000,C 90.000,E1 145.801} C_DIS
LIN {X 0.141,Y -458.985,Z 235.601,A 0.000,B 0.000,C 90.000,E1 144.196} C_DIS
LIN {X -0.151,Y -461.539,Z 235.592,A 0.000,B 0.000,C 90.000,E1 142.637} C_DIS
LIN {X 0.168,Y -463.820,Z 235.584,A 0.000,B 0.000,C 90.000,E1 141.009} C_DIS
LIN {X 0.129,Y -465.442,Z 235.577,A 0.000,B 0.000,C 90.000,E1 139.747} C_DIS
LIN {X 0.172,Y -467.289,Z 235.568,A 0.000,B 0.000,C 90.000,E1 138.162} C_DIS
LIN {X 0.139,Y -468.330,Z 235.561,A 0.000,B 0.000,C 90.000,E1 136.905} C_DIS
LIN {X 0.121,Y -469.096,Z 235.554,A 0.000,B 0.000,C 90.000,E1 135.648} C_DIS
LIN {X -0.222,Y -469.645,Z 235.547,A 0.000,B 0.000,C 90.000,E1 134.433} C_DIS
LIN {X 0.021,Y -469.799,Z 235.542,A 0.000,B 0.000,C 90.000,E1 133.461} C_DIS
LIN {X 0.020,Y -469.536,Z 235.535,A 0.000,B 0.000,C 90.000,E1 132.204} C_DIS
LIN {X 0.126,Y -468.722,Z 235.526,A 0.000,B 0.000,C 90.000,E1 130.620} C_DIS
LIN {X -0.272,Y -468.179,Z 235.521,A 0.000,B 0.000,C 90.000,E1 129.725} C_DIS
LIN {X 0.168,Y -466.922,Z 235.512,A 0.000,B 0.000,C 90.000,E1 128.096} C_DIS
LIN {X -0.124,Y -465.693,Z 235.505,A 0.000,B 0.000,C 90.000,E1 126.870} C_DIS
LIN {X 0.183,Y -464.518,Z 235.500,A 0.000,B 0.000,C 90.000,E1 125.884} C_DIS
LIN {X 0.228,Y -462.782,Z 235.492,A 0.000,B 0.000,C 90.000,E1 124.612} C_DIS
LIN {X -0.018,Y -460.880,Z 235.485,A 0.000,B 0.000,C 90.000,E1 123.372} C_DIS
LIN {X 0.096,Y -458.801,Z 235.478,A 0.000,B 0.000,C 90.000,E1 122.084} C_DIS
LIN {X -0.107,Y -456.099,Z 235.469,A 0.000,B 0.000,C 90.000,E1 120.512} C_DIS
LIN {X 0.086,Y -453.867,Z 235.462,A 0.000,B 0.000,C 90.000,E1 119.205} C_DIS
LIN {X 0.122,Y -450.961,Z 235.453,A 0.000,B 0.000,C 90.000,E1 117.590} C_DIS
LIN {X -0.027,Y -447.479,Z 235.443,A 0.000,B 0.000,C 90.000,E1 115.668} C_DIS
LIN {X -0.074,Y -445.572,Z 235.436,A 0.000,B 0.000,C 90.000,E1 114.567} C_DIS
LIN {X -0.113,Y -445.577,Z 235.436,A 0.000,B 0.000,C 90.000,E1 114.567} C_DIS
LIN {X 0.068,Y -454.515,Z 235.416,A 0.000,B 0.000,C 90.000,E1 110.791} C_DIS
LIN {X 0.187,Y -457.188,Z 235.410,A 0.000,B 0.000,C 90.000,E1 109.812} C_DIS
LIN {X 0.053,Y -466.581,Z 235.385,A 0.000,B 0.000,C 90.000,E1 105.371} C_DIS
LIN {X -0.024,Y -467.369,Z 235.384,A 0.000,B 0.000,C 90.000,E1 105.064} C_DIS
LIN {X -0.220,Y -468.017,Z 235.382,A 0.000,B 0.000,C 90.000,E1 104.773} C_DIS
LIN {X 0.211,Y -476.231,Z 235.356,A 0.000,B 0.000,C 90.000,E1 100.018} C_DIS
LIN {X -0.004,Y -482.127,Z 235.330,A 0.000,B 0.000,C 90.000,E1 95.391} C_DIS
LIN {X 0.231,Y -485.527,Z 235.304,A 0.000,B 0.000,C 90.000,E1 90.745} C_DIS
LIN {X -0.222,Y -486.381,Z 235.280,A 0.000,B 0.000,C 90.000,E1 86.502} C_DIS
LIN {X 0.088,Y -486.352,Z 235.279,A 0.000,B 0.000,C 90.000,E1 86.159} C_DIS
LIN {X 0.166,Y -484.667,Z 235.253,A 0.000,B 0.000,C 90.000,E1 81.546} C_DIS
LIN {X 0.055,Y -480.586,Z 235.228,A 0.000,B 0.000,C 90.000,E1 76.937} C_DIS
LIN {X -0.231,Y -479.667,Z 235.224,A 0.000,B 0.000,C 90.000,E1 76.353} C_DIS
LIN {X -0.197,Y -474.007,Z 235.200,A 0.000,B 0.000,C 90.000,E1 72.000} C_DIS
LIN {X -0.053,Y -466.365,Z 235.176,A 0.000,B 0.000,C 90.000,E1 67.592} C_DIS
LIN {X -0.166,Y -465.419,Z 235.172,A 0.000,B 0.000,C 90.000,E1 66.975} C_DIS
LIN {X 0.082,Y -461.215,Z 235.161,A 0.000,B 0.000,C 90.000,E1 65.049} C_DIS
LIN {X 0.042,Y -461.223,Z 235.161,A 0.000,B 0.000,C 90.000,E1 65.049} C_DIS
LIN {X 0.090,Y -465.635,Z 235.152,A 0.000,B 0.000,C 90.000,E1 63.332} C_DIS
LIN {X -0.260,Y -467.189,Z 235.148,A 0.000,B 0.000,C 90.000,E1 62.743} C_DIS
LIN {X -0.030,Y -469.774,Z 235.143,A 0.000,B 0.000,C 90.000,E1 61.769} C_DIS
LIN {X -0.011,Y -473.059,Z 235.136,A 0.000,B 0.000,C 90.000,E1 60.511} C_DIS
LIN {X -0.122,Y -475.524,Z 235.131,A 0.000,B 0.000,C 90.000,E1 59.587} C_DIS
LIN {X 0.064,Y -476.238,Z 235.129,A 0.000,B 0.000,C 90.000,E1 59.253} C_DIS
LIN {X 0.020,Y -478.810,Z 235.124,A 0.000,B 0.000,C 90.000,E1 58.329} C_DIS
LIN {X -0.026,Y -483.114,Z 235.116,A 0.000,B 0.000,C 90.000,E1 56.786} C_DIS
LIN {X 0.228,Y -484.099,Z 235.113,A 0.000,B 0.000,C 90.000,E1 56.294} C_DIS
LIN {X -0.160,Y -485.218,Z 235.111,A 0.000,B 0.000,C 90.000,E1 56.008} C_DIS
LIN {X 0.112,Y -487.484,Z 235.106,A 0.000,B 0.000,C 90.000,E1 55.055} C_DIS
LIN {X 0.131,Y -490.336,Z 235.099,A 0.000,B 0.000,C 90.000,E1 53.829} C_DIS
LIN {X -0.098,Y -493.048,Z 235.092,A 0.000,B 0.000,C 90.000,E1 52.637} C_DIS
LIN {X 0.004,Y -495.442,Z 235.086,A 0.000,B 0.000,C 90.000,E1 51.412} C_DIS
LIN {X 0.070,Y -497.478,Z 235.079,A 0.000,B 0.000,C 90.000,E1 50.194} C_DIS
LIN {X -0.151,Y -499.331,Z 235.072,A 0.000,B 0.000,C 90.000,E1 49.013} C_DIS
LIN {X 0.111,Y -500.608,Z 235.067,A 0.000,B 0.000,C 90.000,E1 48.081} C_DIS
LIN {X -0.110,Y -501.992,Z 235.061,A 0.000,B 0.000,C 90.000,E1 46.905} C_DIS
LIN {X -0.312,Y -503.119,Z 235.054,A 0.000,B 0.000,C 90.000,E1 45.729} C_DIS
LIN {X -0.013,Y -503.708,Z 235.049,A 0.000,B 0.000,C 90.000,E1 44.798} C_DIS
LIN {X -0.198,Y -504.147,Z 235.042,A 0.000,B 0.000,C 90.000,E1 43.623} C_DIS
LIN {X 0.119,Y -504.289,Z 235.037,A 0.000,B 0.000,C 90.000,E1 42.690} C_DIS
LIN {X -0.055,Y -504.040,Z 235.031,A 0.000,B 0.000,C 90.000,E1 41.515} C_DIS
LIN {X -0.072,Y -503.755,Z 235.026,A 0.000,B 0.000,C 90.000,E1 40.620} C_DIS
LIN {X 0.004,Y -502.879,Z 235.017,A 0.000,B 0.000,C 90.000,E1 39.116} C_DIS
LIN {X -0.028,Y -502.108,Z 235.012,A 0.000,B 0.000,C 90.000,E1 38.222} C_DIS
LIN {X 0.083,Y -500.259,Z 235.004,A 0.000,B 0.000,C 90.000,E1 36.710} C_DIS
LIN {X -0.138,Y -497.984,Z 234.996,A 0.000,B 0.000,C 90.000,E1 35.231} C_DIS
LIN {X 0.010,Y -495.394,Z 234.987,A 0.000,B 0.000,C 90.000,E1 33.706} C_DIS
LIN {X -0.068,Y -488.237,Z 234.964,A 0.000,B 0.000,C 90.000,E1 29.461} C_DIS
LIN {X 0.246,Y -484.370,Z 234.947,A 0.000,B 0.000,C 90.000,E1 26.360} C_DIS
LIN {X 0.032,Y -483.270,Z 234.940,A 0.000,B 0.000,C 90.000,E1 25.155} C_DIS
LIN {X -0.195,Y -481.859,Z 234.930,A 0.000,B 0.000,C 90.000,E1 23.334} C_DIS
LIN {X -0.035,Y -479.818,Z 234.916,A 0.000,B 0.000,C 90.000,E1 20.844} C_DIS
LIN {X -0.026,Y -477.579,Z 234.900,A 0.000,B 0.000,C 90.000,E1 18.055} C_DIS
LIN {X -0.146,Y -476.161,Z 234.890,A 0.000,B 0.000,C 90.000,E1 16.205} C_DIS
LIN {X 0.163,Y -474.931,Z 234.880,A 0.000,B 0.000,C 90.000,E1 14.300} C_DIS
LIN {X -0.184,Y -473.378,Z 234.864,A 0.000,B 0.000,C 90.000,E1 11.535} C_DIS
LIN {X 0.200,Y -472.639,Z 234.854,A 0.000,B 0.000,C 90.000,E1 9.613} C_DIS
LIN {X 0.199,Y -472.134,Z 234.845,A 0.000,B 0.000,C 90.000,E1 8.049} C_DIS
LIN {X -0.050,Y -471.692,Z 234.834,A 0.000,B 0.000,C 90.000,E1 6.201} C_DIS
LIN {X 0.112,Y -471.512,Z 234.824,A 0.000,B 0.000,C 90.000,E1 4.302} C_DIS
LIN {X -0.012,Y -471.597,Z 234.815,A 0.000,B 0.000,C 90.000,E1 2.751} C_DIS
LIN {X 0.214,Y -472.527,Z 234.795,A 0.000,B 0.000,C 90.000,E1 359.141} C_DIS
LIN {X -0.068,Y -474.046,Z 234.782,A 0.000,B 0.000,C 90.000,E1 356.674} C_DIS
LIN {X -0.054,Y -475.672,Z 234.769,A 0.000,B 0.000,C 90.000,E1 354.489} C_DIS
LIN {X -0.171,Y -479.409,Z 234.750,A 0.000,B 0.000,C 90.000,E1 351.084} C_DIS
LIN {X 0.189,Y -481.307,Z 234.744,A 0.000,B 0.000,C 90.000,E1 349.803} C_DIS
LIN {X 0.191,Y -485.922,Z 234.732,A 0.000,B 0.000,C 90.000,E1 347.645} C_DIS
LIN {X -0.055,Y -492.415,Z 234.718,A 0.000,B 0.000,C 90.000,E1 345.227} C_DIS
LIN {X 0.201,Y -497.299,Z 234.708,A 0.000,B 0.000,C 90.000,E1 343.378} C_DIS
LIN {X 0.151,Y -504.829,Z 234.693,A 0.000,B 0.000,C 90.000,E1 340.678} C_DIS
LIN {X 0.147,Y -515.139,Z 234.675,A 0.000,B 0.000,C 90.000,E1 337.411} C_DIS
LIN {X 0.150,Y -522.280,Z 234.663,A 0.000,B 0.000,C 90.000,E1 335.357} C_DIS
LIN {X 0.066,Y -529.551,Z 234.652,A 0.000,B 0.000,C 90.000,E1 333.332} C_DIS
LIN {X 0.311,Y -533.906,Z 234.646,A 0.000,B 0.000,C 90.000,E1 332.153} C_DIS
LIN {X 0.092,Y -539.333,Z 234.638,A 0.000,B 0.000,C 90.000,E1 330.745} C_DIS
LIN {X 0.013,Y -543.567,Z 234.631,A 0.000,B 0.000,C 90.000,E1 329.616} C_DIS
LIN {X -0.186,Y -550.857,Z 234.620,A 0.000,B 0.000,C 90.000,E1 327.661} C_DIS
LIN {X 0.097,Y -558.209,Z 234.609,A 0.000,B 0.000,C 90.000,E1 325.674} C_DIS
LIN {X 0.221,Y -563.536,Z 234.602,A 0.000,B 0.000,C 90.000,E1 324.276} C_DIS
LIN {X -0.020,Y -568.708,Z 234.594,A 0.000,B 0.000,C 90.000,E1 322.924} C_DIS
LIN {X 0.173,Y -573.585,Z 234.586,A 0.000,B 0.000,C 90.000,E1 321.537} C_DIS
LIN {X -0.167,Y -585.664,Z 234.568,A 0.000,B 0.000,C 90.000,E1 318.324} C_DIS
LIN {X -0.171,Y -591.258,Z 234.561,A 0.000,B 0.000,C 90.000,E1 316.986} C_DIS
LIN {X -0.077,Y -596.273,Z 234.554,A 0.000,B 0.000,C 90.000,E1 315.648} C_DIS
LIN {X -0.114,Y -599.743,Z 234.548,A 0.000,B 0.000,C 90.000,E1 314.595} C_DIS
LIN {X 0.100,Y -601.988,Z 234.543,A 0.000,B 0.000,C 90.000,E1 313.785} C_DIS
LIN {X -0.078,Y -604.001,Z 234.539,A 0.000,B 0.000,C 90.000,E1 313.014} C_DIS
LIN {X 0.175,Y -605.673,Z 234.535,A 0.000,B 0.000,C 90.000,E1 312.204} C_DIS
LIN {X 0.034,Y -607.117,Z 234.530,A 0.000,B 0.000,C 90.000,E1 311.434} C_DIS
LIN {X 0.172,Y -608.622,Z 234.524,A 0.000,B 0.000,C 90.000,E1 310.378} C_DIS
LIN {X -0.252,Y -610.272,Z 234.517,A 0.000,B 0.000,C 90.000,E1 309.116} C_DIS
LIN {X 0.025,Y -611.434,Z 234.511,A 0.000,B 0.000,C 90.000,E1 308.051} C_DIS
LIN {X -0.160,Y -612.373,Z 234.506,A 0.000,B 0.000,C 90.000,E1 307.030} C_DIS
LIN {X 0.158,Y -612.931,Z 234.500,A 0.000,B 0.000,C 90.000,E1 305.964} C_DIS
LIN {X -0.023,Y -613.347,Z 234.494,A 0.000,B 0.000,C 90.000,E1 304.945} C_DIS
LIN {X -0.102,Y -613.619,Z 234.487,A 0.000,B 0.000,C 90.000,E1 303.658} C_DIS
LIN {X -0.080,Y -613.491,Z 234.483,A 0.000,B 0.000,C 90.000,E1 302.880} C_DIS
LIN {X -0.156,Y -612.490,Z 234.475,A 0.000,B 0.000,C 90.000,E1 301.592} C_DIS
LIN {X 0.268,Y -610.727,Z 234.468,A 0.000,B 0.000,C 90.000,E1 300.256} C_DIS
LIN {X -0.177,Y -608.341,Z 234.461,A 0.000,B 0.000,C 90.000,E1 298.999} C_DIS
LIN {X -0.318,Y -606.751,Z 234.457,A 0.000,B 0.000,C 90.000,E1 298.231} C_DIS
LIN {X 0.294,Y -604.349,Z 234.451,A 0.000,B 0.000,C 90.000,E1 297.129} C_DIS
LIN {X 0.057,Y -601.841,Z 234.445,A 0.000,B 0.000,C 90.000,E1 296.104} C_DIS
LIN {X 0.174,Y -597.746,Z 234.436,A 0.000,B 0.000,C 90.000,E1 294.515} C_DIS
LIN {X -0.021,Y -591.795,Z 234.423,A 0.000,B 0.000,C 90.000,E1 292.153} C_DIS
LIN {X 0.303,Y -588.812,Z 234.416,A 0.000,B 0.000,C 90.000,E1 290.791} C_DIS
LIN {X -0.112,Y -584.815,Z 234.405,A 0.000,B 0.000,C 90.000,E1 288.960} C_DIS
LIN {X 0.244,Y -582.041,Z 234.398,A 0.000,B 0.000,C 90.000,E1 287.583} C_DIS
LIN {X 0.242,Y -577.806,Z 234.386,A 0.000,B 0.000,C 90.000,E1 285.426} C_DIS
LIN {X 0.022,Y -573.581,Z 234.372,A 0.000,B 0.000,C 90.000,E1 283.008} C_DIS
LIN {X 0.106,Y -569.074,Z 234.354,A 0.000,B 0.000,C 90.000,E1 279.726} C_DIS
LIN {X 0.145,Y -566.672,Z 234.342,A 0.000,B 0.000,C 90.000,E1 277.530} C_DIS
LIN {X -0.217,Y -563.677,Z 234.311,A 0.000,B 0.000,C 90.000,E1 272.064} C_DIS
LIN {X 0.053,Y -564.039,Z 234.291,A 0.000,B 0.000,C 90.000,E1 268.453} C_DIS
LIN {X -0.193,Y -568.715,Z 234.259,A 0.000,B 0.000,C 90.000,E1 262.704} C_DIS
LIN {X 0.159,Y -571.863,Z 234.246,A 0.000,B 0.000,C 90.000,E1 260.208} C_DIS
LIN {X 0.312,Y -574.721,Z 234.235,A 0.000,B 0.000,C 90.000,E1 258.285} C_DIS
LIN {X -0.128,Y -577.389,Z 234.226,A 0.000,B 0.000,C 90.000,E1 256.700} C_DIS
LIN {X -0.038,Y -579.381,Z 234.219,A 0.000,B 0.000,C 90.000,E1 255.338} C_DIS
LIN {X -0.131,Y -580.915,Z 234.213,A 0.000,B 0.000,C 90.000,E1 254.267} C_DIS
LIN {X -0.205,Y -582.350,Z 234.207,A 0.000,B 0.000,C 90.000,E1 253.196} C_DIS
LIN {X 0.069,Y -583.148,Z 234.202,A 0.000,B 0.000,C 90.000,E1 252.362} C_DIS
LIN {X -0.209,Y -583.656,Z 234.198,A 0.000,B 0.000,C 90.000,E1 251.583} C_DIS
LIN {X 0.256,Y -583.867,Z 234.193,A 0.000,B 0.000,C 90.000,E1 250.732} C_DIS
LIN {X -0.166,Y -583.946,Z 234.187,A 0.000,B 0.000,C 90.000,E1 249.699} C_DIS
LIN {X 0.103,Y -583.910,Z 234.184,A 0.000,B 0.000,C 90.000,E1 249.135} C_DIS
LIN {X 0.029,Y -583.539,Z 234.180,A 0.000,B 0.000,C 90.000,E1 248.337} C_DIS
LIN {X 0.083,Y -583.189,Z 234.177,A 0.000,B 0.000,C 90.000,E1 247.794} C_DIS
LIN {X -0.278,Y -581.748,Z 234.169,A 0.000,B 0.000,C 90.000,E1 246.485} C_DIS
LIN {X -0.017,Y -580.812,Z 234.166,A 0.000,B 0.000,C 90.000,E1 245.921} C_DIS
LIN {X 0.239,Y -580.038,Z 234.163,A 0.000,B 0.000,C 90.000,E1 245.357} C_DIS
LIN {X 0.203,Y -577.861,Z 234.157,A 0.000,B 0.000,C 90.000,E1 244.280} C_DIS
LIN {X -0.086,Y -576.470,Z 234.154,A 0.000,B 0.000,C 90.000,E1 243.768} C_DIS
LIN {X -0.233,Y -575.986,Z 234.153,A 0.000,B 0.000,C 90.000,E1 243.512} C_DIS
LIN {X -0.021,Y -574.578,Z 234.150,A 0.000,B 0.000,C 90.000,E1 242.948} C_DIS
LIN {X -0.066,Y -573.324,Z 234.147,A 0.000,B 0.000,C 90.000,E1 242.410} C_DIS
LIN {X -0.223,Y -572.509,Z 234.145,A 0.000,B 0.000,C 90.000,E1 242.153} C_DIS
LIN {X -0.042,Y -571.143,Z 234.142,A 0.000,B 0.000,C 90.000,E1 241.591} C_DIS
LIN {X -0.275,Y -568.815,Z 234.138,A 0.000,B 0.000,C 90.000,E1 240.795} C_DIS
LIN {X -0.026,Y -564.020,Z 234.129,A 0.000,B 0.000,C 90.000,E1 239.125} C_DIS
LIN {X -0.125,Y -562.288,Z 234.125,A 0.000,B 0.000,C 90.000,E1 238.584} C_DIS
LIN {X 0.152,Y -561.511,Z 234.124,A 0.000,B 0.000,C 90.000,E1 238.280} C_DIS
LIN {X 0.032,Y -559.716,Z 234.121,A 0.000,B 0.000,C 90.000,E1 237.740} C_DIS
LIN {X 0.118,Y -558.978,Z 234.119,A 0.000,B 0.000,C 90.000,E1 237.454} C_DIS
LIN {X -0.018,Y -557.120,Z 234.116,A 0.000,B 0.000,C 90.000,E1 236.914} C_DIS
LIN {X 0.139,Y -555.461,Z 234.113,A 0.000,B 0.000,C 90.000,E1 236.342} C_DIS
LIN {X -0.196,Y -551.917,Z 234.107,A 0.000,B 0.000,C 90.000,E1 235.261} C_DIS
LIN {X -0.132,Y -550.917,Z 234.105,A 0.000,B 0.000,C 90.000,E1 234.975} C_DIS
LIN {X -0.011,Y -549.270,Z 234.102,A 0.000,B 0.000,C 90.000,E1 234.402} C_DIS
LIN {X 0.045,Y -548.218,Z 234.101,A 0.000,B 0.000,C 90.000,E1 234.116} C_DIS
LIN {X 0.149,Y -546.582,Z 234.098,A 0.000,B 0.000,C 90.000,E1 233.543} C_DIS
LIN {X 0.019,Y -542.047,Z 234.090,A 0.000,B 0.000,C 90.000,E1 232.145} C_DIS
LIN {X 0.047,Y -541.084,Z 234.088,A 0.000,B 0.000,C 90.000,E1 231.859} C_DIS
LIN {X 0.007,Y -539.501,Z 234.085,A 0.000,B 0.000,C 90.000,E1 231.295} C_DIS
LIN {X 0.061,Y -535.866,Z 234.079,A 0.000,B 0.000,C 90.000,E1 230.150} C_DIS
LIN {X 0.001,Y -533.913,Z 234.076,A 0.000,B 0.000,C 90.000,E1 229.585} C_DIS
LIN {X -0.012,Y -532.154,Z 234.072,A 0.000,B 0.000,C 90.000,E1 229.013} C_DIS
LIN {X -0.238,Y -526.501,Z 234.063,A 0.000,B 0.000,C 90.000,E1 227.310} C_DIS
LIN {X -0.034,Y -523.724,Z 234.058,A 0.000,B 0.000,C 90.000,E1 226.419} C_DIS
LIN {X 0.073,Y -519.902,Z 234.051,A 0.000,B 0.000,C 90.000,E1 225.243} C_DIS
LIN {X -0.002,Y -519.011,Z 234.050,A 0.000,B 0.000,C 90.000,E1 224.960} C_DIS
LIN {X -0.247,Y -516.083,Z 234.045,A 0.000,B 0.000,C 90.000,E1 224.109} C_DIS
LIN {X -0.056,Y -514.370,Z 234.042,A 0.000,B 0.000,C 90.000,E1 223.500} C_DIS
LIN {X 0.009,Y -511.414,Z 234.037,A 0.000,B 0.000,C 90.000,E1 222.609} C_DIS
LIN {X 0.168,Y -509.737,Z 234.033,A 0.000,B 0.000,C 90.000,E1 222.000} C_DIS
LIN {X 0.063,Y -506.001,Z 234.027,A 0.000,B 0.000,C 90.000,E1 220.825} C_DIS
LIN {X -0.148,Y -504.350,Z 234.024,A 0.000,B 0.000,C 90.000,E1 220.253} C_DIS
LIN {X 0.044,Y -500.736,Z 234.017,A 0.000,B 0.000,C 90.000,E1 219.036} C_DIS
LIN {X -0.011,Y -498.278,Z 234.012,A 0.000,B 0.000,C 90.000,E1 218.141} C_DIS
LIN {X 0.272,Y -493.254,Z 234.002,A 0.000,B 0.000,C 90.000,E1 216.297} C_DIS
LIN {X 0.001,Y -487.280,Z 233.990,A 0.000,B 0.000,C 90.000,E1 214.199} C_DIS
LIN {X 0.122,Y -483.849,Z 233.983,A 0.000,B 0.000,C 90.000,E1 212.959} C_DIS
LIN {X -0.057,Y -478.715,Z 233.973,A 0.000,B 0.000,C 90.000,E1 211.131} C_DIS
LIN {X -0.007,Y -469.311,Z 233.952,A 0.000,B 0.000,C 90.000,E1 207.385} C_DIS
LIN {X 0.260,Y -465.278,Z 233.942,A 0.000,B 0.000,C 90.000,E1 205.463} C_DIS
LIN {X 0.044,Y -461.512,Z 233.931,A 0.000,B 0.000,C 90.000,E1 203.590} C_DIS
LIN {X -0.168,Y -458.559,Z 233.922,A 0.000,B 0.000,C 90.000,E1 202.025} C_DIS
LIN {X 0.150,Y -455.416,Z 233.912,A 0.000,B 0.000,C 90.000,E1 200.066} C_DIS
LIN {X -0.240,Y -451.152,Z 233.896,A 0.000,B 0.000,C 90.000,E1 197.221} C_DIS
LIN {X -0.215,Y -448.149,Z 233.883,A 0.000,B 0.000,C 90.000,E1 194.954} C_DIS
LIN {X 0.023,Y -446.129,Z 233.874,A 0.000,B 0.000,C 90.000,E1 193.300} C_DIS
LIN {X 0.111,Y -443.317,Z 233.861,A 0.000,B 0.000,C 90.000,E1 191.007} C_DIS
LIN {X 0.218,Y -441.046,Z 233.850,A 0.000,B 0.000,C 90.000,E1 189.029} C_DIS
LIN {X 0.054,Y -439.355,Z 233.841,A 0.000,B 0.000,C 90.000,E1 187.409} C_DIS
LIN {X -0.099,Y -437.489,Z 233.830,A 0.000,B 0.000,C 90.000,E1 185.454} C_DIS
LIN {X 0.150,Y -435.881,Z 233.819,A 0.000,B 0.000,C 90.000,E1 183.440} C_DIS
LIN {X -0.020,Y -434.119,Z 233.806,A 0.000,B 0.000,C 90.000,E1 181.146} C_DIS
LIN {X -0.077,Y -432.301,Z 233.790,A 0.000,B 0.000,C 90.000,E1 178.165} C_DIS
LIN {X -0.147,Y -431.170,Z 233.773,A 0.000,B 0.000,C 90.000,E1 175.179} C_DIS
LIN {X -0.045,Y -431.101,Z 233.762,A 0.000,B 0.000,C 90.000,E1 173.166} C_DIS
LIN {X -0.155,Y -431.388,Z 233.749,A 0.000,B 0.000,C 90.000,E1 170.849} C_DIS
LIN {X -0.152,Y -432.531,Z 233.725,A 0.000,B 0.000,C 90.000,E1 166.520} C_DIS
LIN {X -0.101,Y -433.376,Z 233.714,A 0.000,B 0.000,C 90.000,E1 164.519} C_DIS
LIN {X -0.144,Y -434.211,Z 233.707,A 0.000,B 0.000,C 90.000,E1 163.196} C_DIS
LIN {X -0.167,Y -434.934,Z 233.699,A 0.000,B 0.000,C 90.000,E1 161.873} C_DIS
LIN {X -0.009,Y -435.465,Z 233.694,A 0.000,B 0.000,C 90.000,E1 160.859} C_DIS
LIN {X 0.124,Y -436.545,Z 233.686,A 0.000,B 0.000,C 90.000,E1 159.518} C_DIS
LIN {X 0.040,Y -439.523,Z 233.668,A 0.000,B 0.000,C 90.000,E1 156.230} C_DIS
LIN {X -0.010,Y -440.854,Z 233.661,A 0.000,B 0.000,C 90.000,E1 154.921} C_DIS
LIN {X 0.144,Y -442.442,Z 233.653,A 0.000,B 0.000,C 90.000,E1 153.589} C_DIS
LIN {X -0.005,Y -446.446,Z 233.637,A 0.000,B 0.000,C 90.000,E1 150.667} C_DIS
LIN {X -0.197,Y -449.487,Z 233.626,A 0.000,B 0.000,C 90.000,E1 148.742} C_DIS
LIN {X 0.251,Y -453.123,Z 233.614,A 0.000,B 0.000,C 90.000,E1 146.421} C_DIS
LIN {X -0.131,Y -455.261,Z 233.607,A 0.000,B 0.000,C 90.000,E1 145.182} C_DIS
LIN {X -0.049,Y -456.448,Z 233.603,A 0.000,B 0.000,C 90.000,E1 144.529} C_DIS
LIN {X -0.016,Y -459.108,Z 233.594,A 0.000,B 0.000,C 90.000,E1 142.924} C_DIS
LIN {X -0.032,Y -461.491,Z 233.585,A 0.000,B 0.000,C 90.000,E1 141.331} C_DIS
LIN {X -0.070,Y -463.611,Z 233.576,A 0.000,B 0.000,C 90.000,E1 139.747} C_DIS
LIN {X -0.064,Y -465.379,Z 233.568,A 0.000,B 0.000,C 90.000,E1 138.162} C_DIS
LIN {X -0.192,Y -466.213,Z 233.562,A 0.000,B 0.000,C 90.000,E1 137.229} C_DIS
LIN {X -0.243,Y -467.052,Z 233.555,A 0.000,B 0.000,C 90.000,E1 135.972} C_DIS
LIN {X 0.043,Y -467.610,Z 233.548,A 0.000,B 0.000,C 90.000,E1 134.676} C_DIS
LIN {X 0.264,Y -467.818,Z 233.543,A 0.000,B 0.000,C 90.000,E1 133.704} C_DIS
LIN {X 0.163,Y -467.759,Z 233.538,A 0.000,B 0.000,C 90.000,E1 132.771} C_DIS
LIN {X 0.062,Y -467.481,Z 233.533,A 0.000,B 0.000,C 90.000,E1 131.838} C_DIS
LIN {X -0.046,Y -466.939,Z 233.527,A 0.000,B 0.000,C 90.000,E1 130.906} C_DIS
LIN {X -0.286,Y -466.847,Z 233.526,A 0.000,B 0.000,C 90.000,E1 130.620} C_DIS
LIN {X 0.008,Y -466.043,Z 233.519,A 0.000,B 0.000,C 90.000,E1 129.322} C_DIS
LIN {X 0.110,Y -464.744,Z 233.510,A 0.000,B 0.000,C 90.000,E1 127.729} C_DIS
LIN {X -0.088,Y -463.066,Z 233.501,A 0.000,B 0.000,C 90.000,E1 126.171} C_DIS
LIN {X 0.067,Y -460.425,Z 233.490,A 0.000,B 0.000,C 90.000,E1 124.246} C_DIS
LIN {X 0.166,Y -458.481,Z 233.483,A 0.000,B 0.000,C 90.000,E1 122.959} C_DIS
LIN {X -0.039,Y -455.860,Z 233.474,A 0.000,B 0.000,C 90.000,E1 121.386} C_DIS
LIN {X -0.144,Y -453.109,Z 233.465,A 0.000,B 0.000,C 90.000,E1 119.795} C_DIS
LIN {X -0.042,Y -449.628,Z 233.455,A 0.000,B 0.000,C 90.000,E1 117.847} C_DIS
LIN {X -0.024,Y -446.178,Z 233.444,A 0.000,B 0.000,C 90.000,E1 115.899} C_DIS
LIN {X -0.203,Y -444.572,Z 233.439,A 0.000,B 0.000,C 90.000,E1 115.027} C_DIS
LIN {X -0.243,Y -444.587,Z 233.439,A 0.000,B 0.000,C 90.000,E1 115.027} C_DIS
LIN {X -0.245,Y -451.417,Z 233.422,A 0.000,B 0.000,C 90.000,E1 112.025} C_DIS
LIN {X -0.149,Y -457.399,Z 233.410,A 0.000,B 0.000,C 90.000,E1 109.758} C_DIS
LIN {X -0.065,Y -466.039,Z 233.387,A 0.000,B 0.000,C 90.000,E1 105.607} C_DIS
LIN {X 0.109,Y -467.608,Z 233.383,A 0.000,B 0.000,C 90.000,E1 104.954} C_DIS
LIN {X 0.106,Y -469.065,Z 233.378,A 0.000,B 0.000,C 90.000,E1 104.008} C_DIS
LIN {X 0.067,Y -475.833,Z 233.357,A 0.000,B 0.000,C 90.000,E1 100.254} C_DIS
LIN {X -0.095,Y -476.319,Z 233.355,A 0.000,B 0.000,C 90.000,E1 99.962} C_DIS
LIN {X -0.148,Y -481.814,Z 233.331,A 0.000,B 0.000,C 90.000,E1 95.625} C_DIS
LIN {X 0.179,Y -482.177,Z 233.329,A 0.000,B 0.000,C 90.000,E1 95.277} C_DIS
LIN {X 0.113,Y -485.324,Z 233.306,A 0.000,B 0.000,C 90.000,E1 90.974} C_DIS
LIN {X -0.062,Y -485.535,Z 233.304,A 0.000,B 0.000,C 90.000,E1 90.688} C_DIS
LIN {X 0.145,Y -486.327,Z 233.282,A 0.000,B 0.000,C 90.000,E1 86.674} C_DIS
LIN {X -0.206,Y -486.294,Z 233.278,A 0.000,B 0.000,C 90.000,E1 86.102} C_DIS
LIN {X -0.001,Y -484.695,Z 233.254,A 0.000,B 0.000,C 90.000,E1 81.781} C_DIS
LIN {X -0.132,Y -484.581,Z 233.253,A 0.000,B 0.000,C 90.000,E1 81.489} C_DIS
LIN {X -0.252,Y -480.519,Z 233.227,A 0.000,B 0.000,C 90.000,E1 76.881} C_DIS
LIN {X 0.112,Y -474.270,Z 233.201,A 0.000,B 0.000,C 90.000,E1 72.181} C_DIS
LIN {X 0.079,Y -473.816,Z 233.199,A 0.000,B 0.000,C 90.000,E1 71.873} C_DIS
LIN {X 0.040,Y -466.234,Z 233.175,A 0.000,B 0.000,C 90.000,E1 67.486} C_DIS
LIN {X -0.018,Y -465.805,Z 233.173,A 0.000,B 0.000,C 90.000,E1 67.177} C_DIS
LIN {X 0.046,Y -464.458,Z 233.170,A 0.000,B 0.000,C 90.000,E1 66.538} C_DIS
LIN {X 0.129,Y -460.445,Z 233.159,A 0.000,B 0.000,C 90.000,E1 64.665} C_DIS
LIN {X 0.090,Y -460.457,Z 233.159,A 0.000,B 0.000,C 90.000,E1 64.665} C_DIS
LIN {X -0.163,Y -462.083,Z 233.156,A 0.000,B 0.000,C 90.000,E1 64.024} C_DIS
LIN {X -0.124,Y -463.461,Z 233.152,A 0.000,B 0.000,C 90.000,E1 63.384} C_DIS
LIN {X 0.004,Y -464.435,Z 233.150,A 0.000,B 0.000,C 90.000,E1 63.050} C_DIS
LIN {X -0.075,Y -465.273,Z 233.149,A 0.000,B 0.000,C 90.000,E1 62.743} C_DIS
LIN {X 0.063,Y -466.309,Z 233.147,A 0.000,B 0.000,C 90.000,E1 62.410} C_DIS
LIN {X -0.198,Y -469.672,Z 233.140,A 0.000,B 0.000,C 90.000,E1 61.179} C_DIS
LIN {X 0.061,Y -472.067,Z 233.135,A 0.000,B 0.000,C 90.000,E1 60.205} C_DIS
LIN {X -0.006,Y -472.965,Z 233.132,A 0.000,B 0.000,C 90.000,E1 59.744} C_DIS
LIN {X -0.004,Y -473.196,Z 233.131,A 0.000,B 0.000,C 90.000,E1 59.587} C_DIS
LIN {X 0.201,Y -474.017,Z 233.129,A 0.000,B 0.000,C 90.000,E1 59.203} C_DIS
LIN {X 0.255,Y -475.440,Z 233.127,A 0.000,B 0.000,C 90.000,E1 58.869} C_DIS
LIN {X 0.150,Y -479.759,Z 233.119,A 0.000,B 0.000,C 90.000,E1 57.327} C_DIS
LIN {X -0.283,Y -480.723,Z 233.116,A 0.000,B 0.000,C 90.000,E1 56.914} C_DIS
LIN {X -0.004,Y -481.820,Z 233.113,A 0.000,B 0.000,C 90.000,E1 56.373} C_DIS
LIN {X 0.304,Y -483.224,Z 233.111,A 0.000,B 0.000,C 90.000,E1 56.008} C_DIS
LIN {X 0.117,Y -484.131,Z 233.110,A 0.000,B 0.000,C 90.000,E1 55.722} C_DIS
LIN {X -0.021,Y -486.225,Z 233.105,A 0.000,B 0.000,C 90.000,E1 54.815} C_DIS
LIN {X 0.202,Y -486.620,Z 233.103,A 0.000,B 0.000,C 90.000,E1 54.482} C_DIS
LIN {X 0.103,Y -487.620,Z 233.101,A 0.000,B 0.000,C 90.000,E1 54.196} C_DIS
LIN {X -0.004,Y -489.749,Z 233.096,A 0.000,B 0.000,C 90.000,E1 53.290} C_DIS
LIN {X 0.129,Y -490.425,Z 233.094,A 0.000,B 0.000,C 90.000,E1 52.970} C_DIS
LIN {X -0.029,Y -490.803,Z 233.093,A 0.000,B 0.000,C 90.000,E1 52.683} C_DIS
LIN {X -0.220,Y -490.755,Z 233.091,A 0.000,B 0.000,C 90.000,E1 52.477} C_DIS
LIN {X 0.128,Y -490.751,Z 233.091,A 0.000,B 0.000,C 90.000,E1 52.431} C_DIS
LIN {X -0.185,Y -491.163,Z 233.091,A 0.000,B 0.000,C 90.000,E1 52.396} C_DIS
LIN {X 0.048,Y -492.107,Z 233.089,A 0.000,B 0.000,C 90.000,E1 52.065} C_DIS
LIN {X 0.047,Y -493.477,Z 233.086,A 0.000,B 0.000,C 90.000,E1 51.457} C_DIS
LIN {X 0.181,Y -496.463,Z 233.076,A 0.000,B 0.000,C 90.000,E1 49.622} C_DIS
LIN {X -0.106,Y -498.209,Z 233.069,A 0.000,B 0.000,C 90.000,E1 48.447} C_DIS
LIN {X -0.245,Y -498.260,Z 233.067,A 0.000,B 0.000,C 90.000,E1 48.162} C_DIS
LIN {X -0.191,Y -499.301,Z 233.064,A 0.000,B 0.000,C 90.000,E1 47.553} C_DIS
LIN {X -0.133,Y -499.975,Z 233.061,A 0.000,B 0.000,C 90.000,E1 46.944} C_DIS
LIN {X -0.228,Y -500.837,Z 233.056,A 0.000,B 0.000,C 90.000,E1 46.053} C_DIS
LIN {X -0.073,Y -500.714,Z 233.055,A 0.000,B 0.000,C 90.000,E1 45.810} C_DIS
LIN {X 0.039,Y -500.979,Z 233.054,A 0.000,B 0.000,C 90.000,E1 45.648} C_DIS
LIN {X -0.252,Y -501.497,Z 233.050,A 0.000,B 0.000,C 90.000,E1 45.081} C_DIS
LIN {X 0.172,Y -501.504,Z 233.047,A 0.000,B 0.000,C 90.000,E1 44.433} C_DIS
LIN {X 0.215,Y -502.029,Z 233.042,A 0.000,B 0.000,C 90.000,E1 43.542} C_DIS
LIN {X -0.202,Y -502.106,Z 233.037,A 0.000,B 0.000,C 90.000,E1 42.690} C_DIS
LIN {X -0.118,Y -502.024,Z 233.034,A 0.000,B 0.000,C 90.000,E1 42.081} C_DIS
LIN {X 0.092,Y -501.733,Z 233.032,A 0.000,B 0.000,C 90.000,E1 41.757} C_DIS
LIN {X -0.032,Y -501.881,Z 233.030,A 0.000,B 0.000,C 90.000,E1 41.472} C_DIS
LIN {X 0.175,Y -501.797,Z 233.029,A 0.000,B 0.000,C 90.000,E1 41.148} C_DIS
LIN {X 0.053,Y -501.499,Z 233.027,A 0.000,B 0.000,C 90.000,E1 40.862} C_DIS
LIN {X -0.019,Y -501.066,Z 233.026,A 0.000,B 0.000,C 90.000,E1 40.744} C_DIS
LIN {X -0.060,Y -501.055,Z 233.026,A 0.000,B 0.000,C 90.000,E1 40.744} C_DIS
LIN {X 0.258,Y -501.404,Z 233.025,A 0.000,B 0.000,C 90.000,E1 40.539} C_DIS
LIN {X 0.134,Y -501.421,Z 233.024,A 0.000,B 0.000,C 90.000,E1 40.253} C_DIS
LIN {X 0.092,Y -500.873,Z 233.019,A 0.000,B 0.000,C 90.000,E1 39.358} C_DIS
LIN {X -0.079,Y -499.665,Z 233.012,A 0.000,B 0.000,C 90.000,E1 38.177} C_DIS
LIN {X -0.148,Y -498.608,Z 233.007,A 0.000,B 0.000,C 90.000,E1 37.282} C_DIS
LIN {X -0.264,Y -496.878,Z 233.000,A 0.000,B 0.000,C 90.000,E1 36.091} C_DIS
LIN {X 0.149,Y -494.463,Z 232.992,A 0.000,B 0.000,C 90.000,E1 34.532} C_DIS
LIN {X -0.043,Y -491.656,Z 232.984,A 0.000,B 0.000,C 90.000,E1 33.038} C_DIS
LIN {X 0.146,Y -489.426,Z 232.977,A 0.000,B 0.000,C 90.000,E1 31.799} C_DIS
LIN {X -0.112,Y -485.252,Z 232.962,A 0.000,B 0.000,C 90.000,E1 29.077} C_DIS
LIN {X 0.102,Y -481.907,Z 232.946,A 0.000,B 0.000,C 90.000,E1 26.283} C_DIS
LIN {X 0.017,Y -479.938,Z 232.932,A 0.000,B 0.000,C 90.000,E1 23.823} C_DIS
LIN {X -0.025,Y -478.738,Z 232.924,A 0.000,B 0.000,C 90.000,E1 22.280} C_DIS
LIN {X -0.118,Y -476.985,Z 232.912,A 0.000,B 0.000,C 90.000,E1 20.120} C_DIS
LIN {X 0.038,Y -475.532,Z 232.901,A 0.000,B 0.000,C 90.000,E1 18.236} C_DIS
LIN {X 0.045,Y -474.384,Z 232.893,A 0.000,B 0.000,C 90.000,E1 16.677} C_DIS
LIN {X -0.149,Y -473.132,Z 232.882,A 0.000,B 0.000,C 90.000,E1 14.828} C_DIS
LIN {X 0.076,Y -471.683,Z 232.868,A 0.000,B 0.000,C 90.000,E1 12.299} C_DIS
LIN {X 0.074,Y -470.665,Z 232.855,A 0.000,B 0.000,C 90.000,E1 9.792} C_DIS
LIN {X -0.040,Y -469.892,Z 232.841,A 0.000,B 0.000,C 90.000,E1 7.296} C_DIS
LIN {X 0.156,Y -469.534,Z 232.827,A 0.000,B 0.000,C 90.000,E1 4.759} C_DIS
LIN {X -0.235,Y -469.637,Z 232.813,A 0.000,B 0.000,C 90.000,E1 2.293} C_DIS
LIN {X 0.032,Y -471.409,Z 232.788,A 0.000,B 0.000,C 90.000,E1 357.593} C_DIS
LIN {X 0.221,Y -473.172,Z 232.776,A 0.000,B 0.000,C 90.000,E1 355.065} C_DIS
LIN {X 0.086,Y -477.396,Z 232.755,A 0.000,B 0.000,C 90.000,E1 351.027} C_DIS
LIN {X -0.059,Y -479.297,Z 232.749,A 0.000,B 0.000,C 90.000,E1 349.803} C_DIS
LIN {X 0.024,Y -483.180,Z 232.740,A 0.000,B 0.000,C 90.000,E1 347.937} C_DIS
LIN {X 0.052,Y -490.450,Z 232.726,A 0.000,B 0.000,C 90.000,E1 345.172} C_DIS
LIN {X 0.153,Y -496.120,Z 232.715,A 0.000,B 0.000,C 90.000,E1 343.032} C_DIS
LIN {X -0.105,Y -505.524,Z 232.699,A 0.000,B 0.000,C 90.000,E1 339.752} C_DIS
LIN {X 0.156,Y -514.151,Z 232.685,A 0.000,B 0.000,C 90.000,E1 337.050} C_DIS
LIN {X -0.131,Y -521.361,Z 232.675,A 0.000,B 0.000,C 90.000,E1 335.025} C_DIS
LIN {X -0.234,Y -528.723,Z 232.665,A 0.000,B 0.000,C 90.000,E1 332.999} C_DIS
LIN {X -0.111,Y -535.297,Z 232.656,A 0.000,B 0.000,C 90.000,E1 331.257} C_DIS
LIN {X -0.246,Y -539.590,Z 232.651,A 0.000,B 0.000,C 90.000,E1 330.127} C_DIS
LIN {X 0.165,Y -544.796,Z 232.643,A 0.000,B 0.000,C 90.000,E1 328.663} C_DIS
LIN {X 0.208,Y -550.043,Z 232.636,A 0.000,B 0.000,C 90.000,E1 327.248} C_DIS
LIN {X -0.055,Y -556.403,Z 232.628,A 0.000,B 0.000,C 90.000,E1 325.595} C_DIS
LIN {X 0.038,Y -561.762,Z 232.621,A 0.000,B 0.000,C 90.000,E1 324.196} C_DIS
LIN {X -0.233,Y -566.966,Z 232.614,A 0.000,B 0.000,C 90.000,E1 322.844} C_DIS
LIN {X 0.063,Y -572.857,Z 232.606,A 0.000,B 0.000,C 90.000,E1 321.170} C_DIS
LIN {X -0.209,Y -583.042,Z 232.592,A 0.000,B 0.000,C 90.000,E1 318.485} C_DIS
LIN {X 0.251,Y -586.306,Z 232.588,A 0.000,B 0.000,C 90.000,E1 317.634} C_DIS
LIN {X -0.263,Y -588.541,Z 232.586,A 0.000,B 0.000,C 90.000,E1 317.148} C_DIS
LIN {X 0.020,Y -592.756,Z 232.580,A 0.000,B 0.000,C 90.000,E1 316.053} C_DIS
LIN {X -0.290,Y -597.318,Z 232.574,A 0.000,B 0.000,C 90.000,E1 314.757} C_DIS
LIN {X -0.317,Y -600.350,Z 232.568,A 0.000,B 0.000,C 90.000,E1 313.704} C_DIS
LIN {X -0.102,Y -602.288,Z 232.564,A 0.000,B 0.000,C 90.000,E1 312.894} C_DIS
LIN {X 0.168,Y -603.907,Z 232.561,A 0.000,B 0.000,C 90.000,E1 312.081} C_DIS
LIN {X -0.238,Y -604.912,Z 232.558,A 0.000,B 0.000,C 90.000,E1 311.595} C_DIS
LIN {X -0.130,Y -606.443,Z 232.553,A 0.000,B 0.000,C 90.000,E1 310.539} C_DIS
LIN {X 0.069,Y -608.415,Z 232.545,A 0.000,B 0.000,C 90.000,E1 308.955} C_DIS
LIN {X 0.038,Y -609.258,Z 232.541,A 0.000,B 0.000,C 90.000,E1 308.177} C_DIS
LIN {X 0.103,Y -610.315,Z 232.534,A 0.000,B 0.000,C 90.000,E1 306.870} C_DIS
LIN {X -0.181,Y -610.968,Z 232.528,A 0.000,B 0.000,C 90.000,E1 305.598} C_DIS
LIN {X 0.108,Y -611.316,Z 232.523,A 0.000,B 0.000,C 90.000,E1 304.532} C_DIS
LIN {X -0.174,Y -611.325,Z 232.520,A 0.000,B 0.000,C 90.000,E1 304.040} C_DIS
LIN {X -0.232,Y -611.484,Z 232.519,A 0.000,B 0.000,C 90.000,E1 303.785} C_DIS
LIN {X -0.284,Y -611.136,Z 232.514,A 0.000,B 0.000,C 90.000,E1 302.752} C_DIS
LIN {X -0.056,Y -610.765,Z 232.511,A 0.000,B 0.000,C 90.000,E1 302.212} C_DIS
LIN {X 0.125,Y -610.051,Z 232.507,A 0.000,B 0.000,C 90.000,E1 301.416} C_DIS
LIN {X -0.176,Y -609.359,Z 232.505,A 0.000,B 0.000,C 90.000,E1 300.924} C_DIS
LIN {X -0.060,Y -607.821,Z 232.499,A 0.000,B 0.000,C 90.000,E1 299.873} C_DIS
LIN {X -0.016,Y -605.369,Z 232.493,A 0.000,B 0.000,C 90.000,E1 298.565} C_DIS
LIN {X 0.103,Y -603.726,Z 232.489,A 0.000,B 0.000,C 90.000,E1 297.769} C_DIS
LIN {X -0.278,Y -599.973,Z 232.481,A 0.000,B 0.000,C 90.000,E1 296.232} C_DIS
LIN {X -0.194,Y -596.032,Z 232.473,A 0.000,B 0.000,C 90.000,E1 294.643} C_DIS
LIN {X -0.010,Y -593.267,Z 232.468,A 0.000,B 0.000,C 90.000,E1 293.567} C_DIS
LIN {X -0.229,Y -588.388,Z 232.457,A 0.000,B 0.000,C 90.000,E1 291.461} C_DIS
LIN {X -0.030,Y -583.221,Z 232.445,A 0.000,B 0.000,C 90.000,E1 289.033} C_DIS
LIN {X -0.071,Y -580.465,Z 232.438,A 0.000,B 0.000,C 90.000,E1 287.692} C_DIS
LIN {X -0.127,Y -576.238,Z 232.428,A 0.000,B 0.000,C 90.000,E1 285.536} C_DIS
LIN {X 0.151,Y -571.964,Z 232.415,A 0.000,B 0.000,C 90.000,E1 283.063} C_DIS
LIN {X 0.182,Y -568.391,Z 232.403,A 0.000,B 0.000,C 90.000,E1 280.602} C_DIS
LIN {X 0.030,Y -566.481,Z 232.395,A 0.000,B 0.000,C 90.000,E1 278.973} C_DIS
LIN {X -0.159,Y -562.712,Z 232.373,A 0.000,B 0.000,C 90.000,E1 274.588} C_DIS
LIN {X 0.274,Y -561.894,Z 232.352,A 0.000,B 0.000,C 90.000,E1 270.401} C_DIS
LIN {X -0.151,Y -562.263,Z 232.343,A 0.000,B 0.000,C 90.000,E1 268.511} C_DIS
LIN {X 0.202,Y -567.177,Z 232.312,A 0.000,B 0.000,C 90.000,E1 262.413} C_DIS
LIN {X -0.148,Y -570.368,Z 232.300,A 0.000,B 0.000,C 90.000,E1 259.982} C_DIS
LIN {X -0.126,Y -572.896,Z 232.292,A 0.000,B 0.000,C 90.000,E1 258.342} C_DIS
LIN {X -0.042,Y -575.538,Z 232.284,A 0.000,B 0.000,C 90.000,E1 256.700} C_DIS
LIN {X 0.018,Y -577.550,Z 232.277,A 0.000,B 0.000,C 90.000,E1 255.338} C_DIS
LIN {X 0.111,Y -579.434,Z 232.270,A 0.000,B 0.000,C 90.000,E1 253.976} C_DIS
LIN {X 0.011,Y -580.773,Z 232.265,A 0.000,B 0.000,C 90.000,E1 252.906} C_DIS
LIN {X -0.291,Y -581.505,Z 232.261,A 0.000,B 0.000,C 90.000,E1 252.127} C_DIS
LIN {X -0.244,Y -581.854,Z 232.258,A 0.000,B 0.000,C 90.000,E1 251.583} C_DIS
LIN {X 0.201,Y -582.031,Z 232.254,A 0.000,B 0.000,C 90.000,E1 250.732} C_DIS
LIN {X -0.245,Y -582.134,Z 232.248,A 0.000,B 0.000,C 90.000,E1 249.699} C_DIS
LIN {X 0.201,Y -581.916,Z 232.244,A 0.000,B 0.000,C 90.000,E1 248.847} C_DIS
LIN {X 0.099,Y -581.510,Z 232.240,A 0.000,B 0.000,C 90.000,E1 248.050} C_DIS
LIN {X -0.295,Y -580.093,Z 232.234,A 0.000,B 0.000,C 90.000,E1 246.741} C_DIS
LIN {X -0.189,Y -578.840,Z 232.230,A 0.000,B 0.000,C 90.000,E1 245.921} C_DIS
LIN {X 0.196,Y -578.569,Z 232.228,A 0.000,B 0.000,C 90.000,E1 245.613} C_DIS
LIN {X 0.138,Y -576.377,Z 232.223,A 0.000,B 0.000,C 90.000,E1 244.537} C_DIS
LIN {X 0.048,Y -573.913,Z 232.217,A 0.000,B 0.000,C 90.000,E1 243.461} C_DIS
LIN {X -0.007,Y -572.505,Z 232.215,A 0.000,B 0.000,C 90.000,E1 242.922} C_DIS
LIN {X -0.166,Y -571.956,Z 232.213,A 0.000,B 0.000,C 90.000,E1 242.666} C_DIS
LIN {X 0.014,Y -570.407,Z 232.211,A 0.000,B 0.000,C 90.000,E1 242.103} C_DIS
LIN {X -0.154,Y -569.802,Z 232.209,A 0.000,B 0.000,C 90.000,E1 241.847} C_DIS
LIN {X 0.193,Y -566.663,Z 232.204,A 0.000,B 0.000,C 90.000,E1 240.717} C_DIS
LIN {X 0.111,Y -561.901,Z 232.195,A 0.000,B 0.000,C 90.000,E1 239.076} C_DIS
LIN {X -0.006,Y -560.212,Z 232.193,A 0.000,B 0.000,C 90.000,E1 238.535} C_DIS
LIN {X 0.079,Y -559.405,Z 232.191,A 0.000,B 0.000,C 90.000,E1 238.250} C_DIS
LIN {X -0.132,Y -558.455,Z 232.190,A 0.000,B 0.000,C 90.000,E1 237.995} C_DIS
LIN {X -0.269,Y -556.829,Z 232.187,A 0.000,B 0.000,C 90.000,E1 237.454} C_DIS
LIN {X 0.253,Y -552.474,Z 232.180,A 0.000,B 0.000,C 90.000,E1 236.008} C_DIS
LIN {X 0.070,Y -550.744,Z 232.177,A 0.000,B 0.000,C 90.000,E1 235.468} C_DIS
LIN {X 0.186,Y -548.753,Z 232.175,A 0.000,B 0.000,C 90.000,E1 234.895} C_DIS
LIN {X 0.240,Y -547.993,Z 232.173,A 0.000,B 0.000,C 90.000,E1 234.609} C_DIS
LIN {X 0.019,Y -546.071,Z 232.170,A 0.000,B 0.000,C 90.000,E1 234.069} C_DIS
LIN {X 0.142,Y -543.478,Z 232.166,A 0.000,B 0.000,C 90.000,E1 233.210} C_DIS
LIN {X -0.193,Y -540.826,Z 232.162,A 0.000,B 0.000,C 90.000,E1 232.396} C_DIS
LIN {X -0.144,Y -538.923,Z 232.159,A 0.000,B 0.000,C 90.000,E1 231.823} C_DIS
LIN {X -0.111,Y -537.265,Z 232.156,A 0.000,B 0.000,C 90.000,E1 231.251} C_DIS
LIN {X -0.161,Y -533.710,Z 232.151,A 0.000,B 0.000,C 90.000,E1 230.114} C_DIS
LIN {X 0.121,Y -528.960,Z 232.143,A 0.000,B 0.000,C 90.000,E1 228.647} C_DIS
LIN {X -0.130,Y -524.254,Z 232.136,A 0.000,B 0.000,C 90.000,E1 227.229} C_DIS
LIN {X 0.278,Y -519.427,Z 232.129,A 0.000,B 0.000,C 90.000,E1 225.729} C_DIS
LIN {X -0.050,Y -515.732,Z 232.123,A 0.000,B 0.000,C 90.000,E1 224.595} C_DIS
LIN {X -0.234,Y -513.730,Z 232.120,A 0.000,B 0.000,C 90.000,E1 224.028} C_DIS
LIN {X 0.199,Y -511.049,Z 232.116,A 0.000,B 0.000,C 90.000,E1 223.095} C_DIS
LIN {X -0.120,Y -508.247,Z 232.111,A 0.000,B 0.000,C 90.000,E1 222.243} C_DIS
LIN {X 0.017,Y -506.506,Z 232.108,A 0.000,B 0.000,C 90.000,E1 221.634} C_DIS
LIN {X -0.240,Y -504.505,Z 232.105,A 0.000,B 0.000,C 90.000,E1 221.067} C_DIS
LIN {X -0.041,Y -501.153,Z 232.099,A 0.000,B 0.000,C 90.000,E1 219.850} C_DIS
LIN {X 0.171,Y -497.623,Z 232.093,A 0.000,B 0.000,C 90.000,E1 218.624} C_DIS
LIN {X 0.217,Y -496.019,Z 232.090,A 0.000,B 0.000,C 90.000,E1 218.016} C_DIS
LIN {X -0.194,Y -493.372,Z 232.086,A 0.000,B 0.000,C 90.000,E1 217.156} C_DIS
LIN {X -0.096,Y -490.153,Z 232.080,A 0.000,B 0.000,C 90.000,E1 215.931} C_DIS
LIN {X -0.047,Y -484.124,Z 232.069,A 0.000,B 0.000,C 90.000,E1 213.785} C_DIS
LIN {X -0.190,Y -481.490,Z 232.064,A 0.000,B 0.000,C 90.000,E1 212.880} C_DIS
LIN {X -0.014,Y -476.417,Z 232.055,A 0.000,B 0.000,C 90.000,E1 211.003} C_DIS
LIN {X 0.039,Y -471.390,Z 232.046,A 0.000,B 0.000,C 90.000,E1 209.127} C_DIS
LIN {X -0.068,Y -467.013,Z 232.036,A 0.000,B 0.000,C 90.000,E1 207.257} C_DIS
LIN {X 0.086,Y -464.237,Z 232.030,A 0.000,B 0.000,C 90.000,E1 205.976} C_DIS
LIN {X -0.042,Y -459.912,Z 232.019,A 0.000,B 0.000,C 90.000,E1 203.770} C_DIS
LIN {X 0.047,Y -456.314,Z 232.009,A 0.000,B 0.000,C 90.000,E1 201.844} C_DIS
LIN {X 0.207,Y -452.764,Z 231.998,A 0.000,B 0.000,C 90.000,E1 199.577} C_DIS
LIN {X 0.150,Y -448.604,Z 231.984,A 0.000,B 0.000,C 90.000,E1 196.677} C_DIS
LIN {X -0.170,Y -445.273,Z 231.971,A 0.000,B 0.000,C 90.000,E1 194.120} C_DIS
LIN {X -0.093,Y -443.236,Z 231.962,A 0.000,B 0.000,C 90.000,E1 192.479} C_DIS
LIN {X 0.106,Y -440.812,Z 231.953,A 0.000,B 0.000,C 90.000,E1 190.489} C_DIS
LIN {X 0.021,Y -437.947,Z 231.939,A 0.000,B 0.000,C 90.000,E1 187.871} C_DIS
LIN {X -0.034,Y -435.682,Z 231.928,A 0.000,B 0.000,C 90.000,E1 185.568} C_DIS
LIN {X 0.169,Y -434.070,Z 231.918,A 0.000,B 0.000,C 90.000,E1 183.555} C_DIS
LIN {X -0.051,Y -432.329,Z 231.906,A 0.000,B 0.000,C 90.000,E1 181.260} C_DIS
LIN {X -0.187,Y -430.371,Z 231.891,A 0.000,B 0.000,C 90.000,E1 178.282} C_DIS
LIN {X 0.020,Y -429.339,Z 231.878,A 0.000,B 0.000,C 90.000,E1 175.584} C_DIS
LIN {X -0.185,Y -429.160,Z 231.873,A 0.000,B 0.000,C 90.000,E1 174.609} C_DIS
LIN {X 0.177,Y -429.214,Z 231.866,A 0.000,B 0.000,C 90.000,E1 173.223} C_DIS
LIN {X 0.017,Y -429.411,Z 231.855,A 0.000,B 0.000,C 90.000,E1 170.905} C_DIS
LIN {X -0.066,Y -429.821,Z 231.843,A 0.000,B 0.000,C 90.000,E1 168.578} C_DIS
LIN {X 0.141,Y -430.469,Z 231.835,A 0.000,B 0.000,C 90.000,E1 166.881} C_DIS
LIN {X -0.064,Y -431.434,Z 231.823,A 0.000,B 0.000,C 90.000,E1 164.574} C_DIS
LIN {X -0.135,Y -432.329,Z 231.816,A 0.000,B 0.000,C 90.000,E1 163.251} C_DIS
LIN {X 0.181,Y -433.840,Z 231.803,A 0.000,B 0.000,C 90.000,E1 160.550} C_DIS
LIN {X 0.057,Y -434.637,Z 231.798,A 0.000,B 0.000,C 90.000,E1 159.571} C_DIS
LIN {X -0.101,Y -437.215,Z 231.783,A 0.000,B 0.000,C 90.000,E1 156.613} C_DIS
